LIN {X 0,Y 432.048,Z 691.549,A -85,B 0,C 180,E1 1876.893,E2 1876.893} C_VEL
LIN {X 0,Y 427.007,Z 688.845,A -85,B 0,C 180,E1 1873.962,E2 1873.962} C_VEL
LIN {X 0,Y 421.871,Z 685.398,A -85,B 0,C 180,E1 1871.198,E2 1871.198} C_VEL
LIN {X 0,Y 415.949,Z 680.769,A -85,B 0,C 180,E1 1868.275,E2 1868.275} C_VEL
LIN {X 0,Y 408.852,Z 676.226,A -85,B 0,C 180,E1 1865.437,E2 1865.437} C_VEL
LIN {X 0,Y 401.513,Z 670.583,A -85,B 0,C 180,E1 1862.571,E2 1862.571} C_VEL
LIN {X 0,Y 392.48,Z 664.405,A -85,B 0,C 180,E1 1859.542,E2 1859.542} C_VEL
LIN {X 0,Y 385.757,Z 659.325,A -85,B 0,C 180,E1 1857.38,E2 1857.38} C_VEL
LIN {X 0,Y 377.479,Z 653.334,A -85,B 0,C 180,E1 1854.92,E2 1854.92} C_VEL
LIN {X 0,Y 370.222,Z 647.787,A -85,B 0,C 180,E1 1852.819,E2 1852.819} C_VEL
LIN {X 0,Y 360.53,Z 640.36,A -85,B 0,C 180,E1 1850.166,E2 1850.166} C_VEL
LIN {X 0,Y 343.918,Z 628.074,A -85,B 0,C 180,E1 1845.661,E2 1845.661} C_VEL
LIN {X 0,Y 325.439,Z 613.418,A -85,B 0,C 180,E1 1839.722,E2 1839.722} C_VEL
LIN {X 0,Y 308.556,Z 596.504,A -85,B 0,C 180,E1 1832.543,E2 1832.543} C_VEL
LIN {X 0,Y 297.297,Z 579.607,A -85,B 0,C 180,E1 1825.499,E2 1825.499} C_VEL
LIN {X 0,Y 291.705,Z 565.731,A -85,B 0,C 180,E1 1820.046,E2 1820.046} C_VEL
LIN {X 0,Y 288.211,Z 547.966,A -85,B 0,C 180,E1 1813.697,E2 1813.697} C_VEL
LIN {X 0,Y 287.479,Z 531.833,A -85,B 0,C 180,E1 1808.551,E2 1808.551} C_VEL
LIN {X 0,Y 287.525,Z 526.14,A -85,B 0,C 180,E1 1806.753,E2 1806.753} C_VEL
LIN {X 0,Y 282.899,Z 545.109,A -85,B 0,C 180,E1 1806.656,E2 1806.656} C_VEL
LIN {X 0,Y 277.004,Z 563.845,A -85,B 0,C 180,E1 1806.576,E2 1806.576} C_VEL
LIN {X 0,Y 268.131,Z 586.178,A -85,B 0,C 180,E1 1806.449,E2 1806.449} C_VEL
LIN {X 0,Y 258.493,Z 605.496,A -85,B 0,C 180,E1 1806.291,E2 1806.291} C_VEL
LIN {X 0,Y 248.85,Z 621.951,A -85,B 0,C 180,E1 1806.106,E2 1806.106} C_VEL
LIN {X 0,Y 238.7,Z 637.021,A -85,B 0,C 180,E1 1805.888,E2 1805.888} C_VEL
LIN {X 0,Y 227.028,Z 652.184,A -85,B 0,C 180,E1 1805.601,E2 1805.601} C_VEL
LIN {X 0,Y 211.531,Z 669.665,A -85,B 0,C 180,E1 1805.153,E2 1805.153} C_VEL
LIN {X 0,Y 195.584,Z 684.873,A -85,B 0,C 180,E1 1804.61,E2 1804.61} C_VEL
LIN {X 0,Y 181.403,Z 696.751,A -85,B 0,C 180,E1 1804.026,E2 1804.026} C_VEL
LIN {X 0,Y 167.242,Z 707.237,A -85,B 0,C 180,E1 1803.335,E2 1803.335} C_VEL
LIN {X 0,Y 152.1,Z 717.119,A -85,B 0,C 180,E1 1802.439,E2 1802.439} C_VEL
LIN {X 0,Y 135.999,Z 726.296,A -85,B 0,C 180,E1 1801.251,E2 1801.251} C_VEL
LIN {X 0,Y 116.977,Z 735.612,A -85,B 0,C 180,E1 1799.404,E2 1799.404} C_VEL
LIN {X 0,Y 95.169,Z 744.266,A -85,B 0,C 180,E1 1796.358,E2 1796.358} C_VEL
LIN {X 0,Y 77.459,Z 749.938,A -85,B 0,C 180,E1 1792.583,E2 1792.583} C_VEL
LIN {X 0,Y 61.505,Z 754.079,A -85,B 0,C 180,E1 1787.237,E2 1787.237} C_VEL
LIN {X 0,Y 45.403,Z 757.356,A -85,B 0,C 180,E1 1777.64,E2 1777.64} C_VEL
LIN {X 0,Y 32.323,Z 759.394,A -85,B 0,C 180,E1 1760.647,E2 1760.647} C_VEL
LIN {X 0,Y 24.775,Z 760.386,A -85,B 0,C 180,E1 1731.295,E2 1731.295} C_VEL
LIN {X 0,Y 23.981,Z 760.637,A -85,B 0,C 180,E1 1707.61,E2 1707.61} C_VEL
LIN {X 0,Y 29.264,Z 759.849,A -85,B 0,C 180,E1 1666.9,E2 1666.9} C_VEL
LIN {X 0,Y 43.719,Z 757.656,A -85,B 0,C 180,E1 1643.835,E2 1643.835} C_VEL
LIN {X 0,Y 59.678,Z 754.493,A -85,B 0,C 180,E1 1633.567,E2 1633.567} C_VEL
LIN {X 0,Y 75.698,Z 750.434,A -85,B 0,C 180,E1 1627.892,E2 1627.892} C_VEL
LIN {X 0,Y 92.221,Z 745.27,A -85,B 0,C 180,E1 1624.167,E2 1624.167} C_VEL
LIN {X 0,Y 109.014,Z 738.948,A -85,B 0,C 180,E1 1621.562,E2 1621.562} C_VEL
LIN {X 0,Y 127.974,Z 730.455,A -85,B 0,C 180,E1 1619.46,E2 1619.46} C_VEL
LIN {X 0,Y 149.077,Z 718.975,A -85,B 0,C 180,E1 1617.766,E2 1617.766} C_VEL
LIN {X 0,Y 165.221,Z 708.639,A -85,B 0,C 180,E1 1616.776,E2 1616.776} C_VEL
LIN {X 0,Y 180.391,Z 697.542,A -85,B 0,C 180,E1 1616.019,E2 1616.019} C_VEL
LIN {X 0,Y 193.558,Z 686.651,A -85,B 0,C 180,E1 1615.467,E2 1615.467} C_VEL
LIN {X 0,Y 207.244,Z 673.885,A -85,B 0,C 180,E1 1614.979,E2 1614.979} C_VEL
LIN {X 0,Y 221.286,Z 658.984,A -85,B 0,C 180,E1 1614.555,E2 1614.555} C_VEL
LIN {X 0,Y 236.67,Z 639.862,A -85,B 0,C 180,E1 1614.159,E2 1614.159} C_VEL
LIN {X 0,Y 247.836,Z 623.56,A -85,B 0,C 180,E1 1613.914,E2 1613.914} C_VEL
LIN {X 0,Y 257.478,Z 607.335,A -85,B 0,C 180,E1 1613.727,E2 1613.727} C_VEL
LIN {X 0,Y 266.102,Z 590.426,A -85,B 0,C 180,E1 1613.582,E2 1613.582} C_VEL
LIN {X 0,Y 274.723,Z 570.258,A -85,B 0,C 180,E1 1613.454,E2 1613.454} C_VEL
LIN {X 0,Y 282.17,Z 547.737,A -85,B 0,C 180,E1 1613.355,E2 1613.355} C_VEL
LIN {X 0,Y 287.057,Z 528.29,A -85,B 0,C 180,E1 1613.262,E2 1613.262} C_VEL
LIN {X 0,Y 287.525,Z 526.239,A -85,B 0,C 180,E1 1613.21,E2 1613.21} C_VEL
LIN {X 0,Y 287.819,Z 543.482,A -85,B 0,C 180,E1 1607.765,E2 1607.765} C_VEL
LIN {X 0,Y 288.88,Z 552.893,A -85,B 0,C 180,E1 1604.615,E2 1604.615} C_VEL
LIN {X 0,Y 289.148,Z 557.425,A -85,B 0,C 180,E1 1603.367,E2 1603.367} C_VEL
LIN {X 0,Y 288.555,Z 571.983,A -85,B 0,C 180,E1 1600.311,E2 1600.311} C_VEL
LIN {X 0,Y 288.986,Z 575.602,A -85,B 0,C 180,E1 1599.21,E2 1599.21} C_VEL
LIN {X 0,Y 294.461,Z 588.788,A -85,B 0,C 180,E1 1593.804,E2 1593.804} C_VEL
LIN {X 0,Y 306.56,Z 606.164,A -85,B 0,C 180,E1 1586.264,E2 1586.264} C_VEL
LIN {X 0,Y 326.692,Z 624.896,A -85,B 0,C 180,E1 1578.042,E2 1578.042} C_VEL
LIN {X 0,Y 345.594,Z 639.205,A -85,B 0,C 180,E1 1572.211,E2 1572.211} C_VEL
LIN {X 0,Y 358.052,Z 648.466,A -85,B 0,C 180,E1 1568.819,E2 1568.819} C_VEL
LIN {X 0,Y 367.67,Z 655.59,A -85,B 0,C 180,E1 1566.161,E2 1566.161} C_VEL
LIN {X 0,Y 375.567,Z 661.712,A -85,B 0,C 180,E1 1563.804,E2 1563.804} C_VEL
LIN {X 0,Y 382.824,Z 666.875,A -85,B 0,C 180,E1 1561.628,E2 1561.628} C_VEL
LIN {X 0,Y 391.869,Z 673.574,A -85,B 0,C 180,E1 1558.628,E2 1558.628} C_VEL
LIN {X 0,Y 397.847,Z 677.754,A -85,B 0,C 180,E1 1556.527,E2 1556.527} C_VEL
LIN {X 0,Y 405.855,Z 683.606,A -85,B 0,C 180,E1 1553.366,E2 1553.366} C_VEL
LIN {X 0,Y 411.419,Z 687.152,A -85,B 0,C 180,E1 1551.052,E2 1551.052} C_VEL
LIN {X 0,Y 416.922,Z 691.474,A -85,B 0,C 180,E1 1548.246,E2 1548.246} C_VEL
LIN {X 0,Y 422.748,Z 695.187,A -85,B 0,C 180,E1 1545.078,E2 1545.078} C_VEL
LIN {X 0,Y 427.046,Z 697.466,A -85,B 0,C 180,E1 1542.438,E2 1542.438} C_VEL
LIN {X 0,Y 430.04,Z 700.241,A -85,B 0,C 180,E1 1539.501,E2 1539.501} C_VEL
LIN {X 0,Y 432.467,Z 702.2,A -85,B 0,C 180,E1 1536.504,E2 1536.504} C_VEL
LIN {X 0,Y 434.033,Z 703.321,A -85,B 0,C 180,E1 1533.698,E2 1533.698} C_VEL
LIN {X 0,Y 434.675,Z 703.705,A -85,B 0,C 180,E1 1531.318,E2 1531.318} C_VEL
LIN {X 0,Y 434.753,Z 703.73,A -85,B 0,C 180,E1 1529.209,E2 1529.209} C_VEL
LIN {X 0,Y 434.141,Z 703.379,A -85,B 0,C 180,E1 1526.567,E2 1526.567} C_VEL
LIN {X 0,Y 432.755,Z 702.403,A -85,B 0,C 180,E1 1523.9,E2 1523.9} C_VEL
LIN {X 0,Y 430.41,Z 700.585,A -85,B 0,C 180,E1 1520.912,E2 1520.912} C_VEL
LIN {X 0,Y 427.67,Z 698.099,A -85,B 0,C 180,E1 1518.129,E2 1518.129} C_VEL
LIN {X 0,Y 425.585,Z 696.698,A -85,B 0,C 180,E1 1516.575,E2 1516.575} C_VEL
LIN {X 0,Y 420.846,Z 694.09,A -85,B 0,C 180,E1 1513.863,E2 1513.863} C_VEL
LIN {X 0,Y 415.089,Z 690.135,A -85,B 0,C 180,E1 1510.782,E2 1510.782} C_VEL
LIN {X 0,Y 409.819,Z 686.049,A -85,B 0,C 180,E1 1508.235,E2 1508.235} C_VEL
LIN {X 0,Y 403.522,Z 682.027,A -85,B 0,C 180,E1 1505.715,E2 1505.715} C_VEL
LIN {X 0,Y 396.127,Z 676.336,A -85,B 0,C 180,E1 1502.818,E2 1502.818} C_VEL
LIN {X 0,Y 387.824,Z 670.716,A -85,B 0,C 180,E1 1500.029,E2 1500.029} C_VEL
LIN {X 0,Y 379.753,Z 664.676,A -85,B 0,C 180,E1 1497.412,E2 1497.412} C_VEL
LIN {X 0,Y 370.334,Z 657.748,A -85,B 0,C 180,E1 1494.626,E2 1494.626} C_VEL
LIN {X 0,Y 362.763,Z 652.047,A -85,B 0,C 180,E1 1492.478,E2 1492.478} C_VEL
LIN {X 0,Y 352.04,Z 643.946,A -85,B 0,C 180,E1 1489.57,E2 1489.57} C_VEL
LIN {X 0,Y 337.286,Z 633.069,A -85,B 0,C 180,E1 1485.356,E2 1485.356} C_VEL
LIN {X 0,Y 318.306,Z 617.899,A -85,B 0,C 180,E1 1478.922,E2 1478.922} C_VEL
LIN {X 0,Y 301.774,Z 600.227,A -85,B 0,C 180,E1 1471.124,E2 1471.124} C_VEL
LIN {X 0,Y 291.405,Z 582.303,A -85,B 0,C 180,E1 1463.455,E2 1463.455} C_VEL
LIN {X 0,Y 286.507,Z 564.729,A -85,B 0,C 180,E1 1456.629,E2 1456.629} C_VEL
LIN {X 0,Y 285.15,Z 548.556,A -85,B 0,C 180,E1 1450.979,E2 1450.979} C_VEL
LIN {X 0,Y 285.221,Z 540.34,A -85,B 0,C 180,E1 1448.275,E2 1448.275} C_VEL
LIN {X 0,Y 279.398,Z 559.7,A -85,B 0,C 180,E1 1448.23,E2 1448.23} C_VEL
LIN {X 0,Y 272.99,Z 576.864,A -85,B 0,C 180,E1 1448.187,E2 1448.187} C_VEL
LIN {X 0,Y 265.088,Z 594.503,A -85,B 0,C 180,E1 1448.113,E2 1448.113} C_VEL
LIN {X 0,Y 254.41,Z 614.476,A -85,B 0,C 180,E1 1447.995,E2 1447.995} C_VEL
LIN {X 0,Y 241.969,Z 633.628,A -85,B 0,C 180,E1 1447.838,E2 1447.838} C_VEL
LIN {X 0,Y 230.504,Z 648.864,A -85,B 0,C 180,E1 1447.667,E2 1447.667} C_VEL
LIN {X 0,Y 218.289,Z 663.113,A -85,B 0,C 180,E1 1447.45,E2 1447.45} C_VEL
LIN {X 0,Y 204.038,Z 677.704,A -85,B 0,C 180,E1 1447.155,E2 1447.155} C_VEL
LIN {X 0,Y 185.207,Z 694.205,A -85,B 0,C 180,E1 1446.668,E2 1446.668} C_VEL
LIN {X 0,Y 168.929,Z 706.362,A -85,B 0,C 180,E1 1446.146,E2 1446.146} C_VEL
LIN {X 0,Y 153.68,Z 716.325,A -85,B 0,C 180,E1 1445.542,E2 1445.542} C_VEL
LIN {X 0,Y 138.45,Z 725.037,A -85,B 0,C 180,E1 1444.793,E2 1444.793} C_VEL
LIN {X 0,Y 121.944,Z 733.227,A -85,B 0,C 180,E1 1443.761,E2 1443.761} C_VEL
LIN {X 0,Y 104.055,Z 740.771,A -85,B 0,C 180,E1 1442.262,E2 1442.262} C_VEL
LIN {X 0,Y 81.983,Z 748.355,A -85,B 0,C 180,E1 1439.508,E2 1439.508} C_VEL
LIN {X 0,Y 61.206,Z 753.69,A -85,B 0,C 180,E1 1435.123,E2 1435.123} C_VEL
LIN {X 0,Y 43.904,Z 757.028,A -85,B 0,C 180,E1 1428.282,E2 1428.282} C_VEL
LIN {X 0,Y 28.709,Z 759.125,A -85,B 0,C 180,E1 1414.881,E2 1414.881} C_VEL
LIN {X 0,Y 17.496,Z 760.209,A -85,B 0,C 180,E1 1380.949,E2 1380.949} C_VEL
LIN {X 0,Y 15.972,Z 760.462,A -85,B 0,C 180,E1 1346.411,E2 1346.411} C_VEL
LIN {X 0,Y 25.073,Z 759.54,A -85,B 0,C 180,E1 1291.228,E2 1291.228} C_VEL
LIN {X 0,Y 41.106,Z 757.478,A -85,B 0,C 180,E1 1273.382,E2 1273.382} C_VEL
LIN {X 0,Y 58.278,Z 754.32,A -85,B 0,C 180,E1 1265.744,E2 1265.744} C_VEL
LIN {X 0,Y 75.014,Z 750.256,A -85,B 0,C 180,E1 1261.692,E2 1261.692} C_VEL
LIN {X 0,Y 91.989,Z 745.091,A -85,B 0,C 180,E1 1259.079,E2 1259.079} C_VEL
LIN {X 0,Y 109.097,Z 738.771,A -85,B 0,C 180,E1 1257.266,E2 1257.266} C_VEL
LIN {X 0,Y 128.311,Z 730.279,A -85,B 0,C 180,E1 1255.811,E2 1255.811} C_VEL
LIN {X 0,Y 149.762,Z 718.71,A -85,B 0,C 180,E1 1254.637,E2 1254.637} C_VEL
LIN {X 0,Y 165.878,Z 708.465,A -85,B 0,C 180,E1 1253.966,E2 1253.966} C_VEL
LIN {X 0,Y 181.137,Z 697.367,A -85,B 0,C 180,E1 1253.453,E2 1253.453} C_VEL
LIN {X 0,Y 195.386,Z 685.587,A -85,B 0,C 180,E1 1253.055,E2 1253.055} C_VEL
LIN {X 0,Y 209.636,Z 672.216,A -85,B 0,C 180,E1 1252.726,E2 1252.726} C_VEL
LIN {X 0,Y 225.922,Z 654.529,A -85,B 0,C 180,E1 1252.414,E2 1252.414} C_VEL
LIN {X 0,Y 239.154,Z 637.56,A -85,B 0,C 180,E1 1252.201,E2 1252.201} C_VEL
LIN {X 0,Y 249.836,Z 621.778,A -85,B 0,C 180,E1 1252.056,E2 1252.056} C_VEL
LIN {X 0,Y 259.498,Z 605.326,A -85,B 0,C 180,E1 1251.942,E2 1251.942} C_VEL
LIN {X 0,Y 269.152,Z 586,A -85,B 0,C 180,E1 1251.851,E2 1251.851} C_VEL
LIN {X 0,Y 278.038,Z 563.678,A -85,B 0,C 180,E1 1251.781,E2 1251.781} C_VEL
LIN {X 0,Y 284.004,Z 544.717,A -85,B 0,C 180,E1 1251.736,E2 1251.736} C_VEL
LIN {X 0,Y 285.262,Z 540.289,A -85,B 0,C 180,E1 1251.687,E2 1251.687} C_VEL
LIN {X 0,Y 285.603,Z 557.971,A -85,B 0,C 180,E1 1245.814,E2 1245.814} C_VEL
LIN {X 0,Y 288.188,Z 572.722,A -85,B 0,C 180,E1 1240.333,E2 1240.333} C_VEL
LIN {X 0,Y 288.986,Z 575.602,A -85,B 0,C 180,E1 1239.21,E2 1239.21} C_VEL
LIN {X 0,Y 289.661,Z 579.828,A -85,B 0,C 180,E1 1237.923,E2 1237.923} C_VEL
LIN {X 0,Y 289.945,Z 593.385,A -85,B 0,C 180,E1 1234.696,E2 1234.696} C_VEL
LIN {X 0,Y 290.85,Z 596.648,A -85,B 0,C 180,E1 1233.57,E2 1233.57} C_VEL
LIN {X 0,Y 303.878,Z 614.937,A -85,B 0,C 180,E1 1225.302,E2 1225.302} C_VEL
LIN {X 0,Y 323.118,Z 632.206,A -85,B 0,C 180,E1 1217.425,E2 1217.425} C_VEL
LIN {X 0,Y 340.313,Z 645.101,A -85,B 0,C 180,E1 1211.982,E2 1211.982} C_VEL
LIN {X 0,Y 352.229,Z 653.841,A -85,B 0,C 180,E1 1208.641,E2 1208.641} C_VEL
LIN {X 0,Y 361.939,Z 661.049,A -85,B 0,C 180,E1 1205.959,E2 1205.959} C_VEL
LIN {X 0,Y 370.883,Z 667.919,A -85,B 0,C 180,E1 1203.306,E2 1203.306} C_VEL
LIN {X 0,Y 378.204,Z 673.214,A -85,B 0,C 180,E1 1201.064,E2 1201.064} C_VEL
LIN {X 0,Y 386.833,Z 679.455,A -85,B 0,C 180,E1 1198.185,E2 1198.185} C_VEL
LIN {X 0,Y 392.024,Z 683.129,A -85,B 0,C 180,E1 1196.343,E2 1196.343} C_VEL
LIN {X 0,Y 399.817,Z 688.818,A -85,B 0,C 180,E1 1193.271,E2 1193.271} C_VEL
LIN {X 0,Y 405.586,Z 692.55,A -85,B 0,C 180,E1 1190.876,E2 1190.876} C_VEL
LIN {X 0,Y 411.197,Z 696.903,A -85,B 0,C 180,E1 1187.986,E2 1187.986} C_VEL
LIN {X 0,Y 416.127,Z 700.078,A -85,B 0,C 180,E1 1185.324,E2 1185.324} C_VEL
LIN {X 0,Y 420.877,Z 702.569,A -85,B 0,C 180,E1 1182.465,E2 1182.465} C_VEL
LIN {X 0,Y 423.868,Z 705.347,A -85,B 0,C 180,E1 1179.581,E2 1179.581} C_VEL
LIN {X 0,Y 426.173,Z 707.229,A -85,B 0,C 180,E1 1176.736,E2 1176.736} C_VEL
LIN {X 0,Y 427.744,Z 708.357,A -85,B 0,C 180,E1 1174.021,E2 1174.021} C_VEL
LIN {X 0,Y 428.485,Z 708.783,A -85,B 0,C 180,E1 1171.471,E2 1171.471} C_VEL
LIN {X 0,Y 428.591,Z 708.826,A -85,B 0,C 180,E1 1169.332,E2 1169.332} C_VEL
LIN {X 0,Y 428.064,Z 708.528,A -85,B 0,C 180,E1 1166.787,E2 1166.787} C_VEL
LIN {X 0,Y 426.74,Z 707.626,A -85,B 0,C 180,E1 1164.083,E2 1164.083} C_VEL
LIN {X 0,Y 424.678,Z 706.092,A -85,B 0,C 180,E1 1161.335,E2 1161.335} C_VEL
LIN {X 0,Y 422.103,Z 703.779,A -85,B 0,C 180,E1 1158.663,E2 1158.663} C_VEL
LIN {X 0,Y 419.943,Z 702.077,A -85,B 0,C 180,E1 1156.929,E2 1156.929} C_VEL
LIN {X 0,Y 414.975,Z 699.413,A -85,B 0,C 180,E1 1154.029,E2 1154.029} C_VEL
LIN {X 0,Y 409.055,Z 695.34,A -85,B 0,C 180,E1 1150.883,E2 1150.883} C_VEL
LIN {X 0,Y 404.155,Z 691.495,A -85,B 0,C 180,E1 1148.472,E2 1148.472} C_VEL
LIN {X 0,Y 396.702,Z 686.692,A -85,B 0,C 180,E1 1145.492,E2 1145.492} C_VEL
LIN {X 0,Y 389.268,Z 681.034,A -85,B 0,C 180,E1 1142.631,E2 1142.631} C_VEL
LIN {X 0,Y 380.718,Z 675.133,A -85,B 0,C 180,E1 1139.776,E2 1139.776} C_VEL
LIN {X 0,Y 373.472,Z 669.733,A -85,B 0,C 180,E1 1137.448,E2 1137.448} C_VEL
LIN {X 0,Y 362.618,Z 661.611,A -85,B 0,C 180,E1 1134.233,E2 1134.233} C_VEL
LIN {X 0,Y 353.23,Z 654.62,A -85,B 0,C 180,E1 1131.638,E2 1131.638} C_VEL
LIN {X 0,Y 343.478,Z 647.441,A -85,B 0,C 180,E1 1128.936,E2 1128.936} C_VEL
LIN {X 0,Y 331.052,Z 638.315,A -85,B 0,C 180,E1 1125.217,E2 1125.217} C_VEL
LIN {X 0,Y 313.378,Z 624.206,A -85,B 0,C 180,E1 1118.944,E2 1118.944} C_VEL
LIN {X 0,Y 297.513,Z 607.186,A -85,B 0,C 180,E1 1111.169,E2 1111.169} C_VEL
LIN {X 0,Y 288.151,Z 590.932,A -85,B 0,C 180,E1 1103.953,E2 1103.953} C_VEL
LIN {X 0,Y 283.874,Z 576.6,A -85,B 0,C 180,E1 1098.057,E2 1098.057} C_VEL
LIN {X 0,Y 282.372,Z 561.035,A -85,B 0,C 180,E1 1092.261,E2 1092.261} C_VEL
LIN {X 0,Y 282.538,Z 554.045,A -85,B 0,C 180,E1 1089.857,E2 1089.857} C_VEL
LIN {X 0,Y 274.984,Z 574.891,A -85,B 0,C 180,E1 1089.847,E2 1089.847} C_VEL
LIN {X 0,Y 267.387,Z 592.153,A -85,B 0,C 180,E1 1089.828,E2 1089.828} C_VEL
LIN {X 0,Y 258.203,Z 609.755,A -85,B 0,C 180,E1 1089.797,E2 1089.797} C_VEL
LIN {X 0,Y 245.472,Z 630.284,A -85,B 0,C 180,E1 1089.732,E2 1089.732} C_VEL
LIN {X 0,Y 232.547,Z 647.67,A -85,B 0,C 180,E1 1089.653,E2 1089.653} C_VEL
LIN {X 0,Y 219.995,Z 662.38,A -85,B 0,C 180,E1 1089.55,E2 1089.55} C_VEL
LIN {X 0,Y 206.736,Z 676.035,A -85,B 0,C 180,E1 1089.417,E2 1089.417} C_VEL
LIN {X 0,Y 190.407,Z 690.745,A -85,B 0,C 180,E1 1089.208,E2 1089.208} C_VEL
LIN {X 0,Y 172.034,Z 704.786,A -85,B 0,C 180,E1 1088.911,E2 1088.911} C_VEL
LIN {X 0,Y 155.701,Z 715.531,A -85,B 0,C 180,E1 1088.572,E2 1088.572} C_VEL
LIN {X 0,Y 139.369,Z 724.861,A -85,B 0,C 180,E1 1088.137,E2 1088.137} C_VEL
LIN {X 0,Y 123.045,Z 732.917,A -85,B 0,C 180,E1 1087.58,E2 1087.58} C_VEL
LIN {X 0,Y 105.716,Z 740.196,A -85,B 0,C 180,E1 1086.792,E2 1086.792} C_VEL
LIN {X 0,Y 84.351,Z 747.59,A -85,B 0,C 180,E1 1085.38,E2 1085.38} C_VEL
LIN {X 0,Y 62.066,Z 753.302,A -85,B 0,C 180,E1 1082.94,E2 1082.94} C_VEL
LIN {X 0,Y 43.992,Z 756.699,A -85,B 0,C 180,E1 1079.275,E2 1079.275} C_VEL
LIN {X 0,Y 26.308,Z 758.948,A -85,B 0,C 180,E1 1071.137,E2 1071.137} C_VEL
LIN {X 0,Y 11.352,Z 760.033,A -85,B 0,C 180,E1 1042.433,E2 1042.433} C_VEL
LIN {X 0,Y 7.979,Z 760.286,A -85,B 0,C 180,E1 982.801,E2 982.801} C_VEL
LIN {X 0,Y 21.572,Z 759.403,A -85,B 0,C 180,E1 913.28,E2 913.28} C_VEL
LIN {X 0,Y 40.013,Z 757.3,A -85,B 0,C 180,E1 901.944,E2 901.944} C_VEL
LIN {X 0,Y 58.033,Z 754.142,A -85,B 0,C 180,E1 897.689,E2 897.689} C_VEL
LIN {X 0,Y 75.38,Z 750.035,A -85,B 0,C 180,E1 895.435,E2 895.435} C_VEL
LIN {X 0,Y 92.483,Z 744.914,A -85,B 0,C 180,E1 894.006,E2 894.006} C_VEL
LIN {X 0,Y 109.791,Z 738.595,A -85,B 0,C 180,E1 893.001,E2 893.001} C_VEL
LIN {X 0,Y 130.185,Z 729.636,A -85,B 0,C 180,E1 892.161,E2 892.161} C_VEL
LIN {X 0,Y 150.597,Z 718.623,A -85,B 0,C 180,E1 891.553,E2 891.553} C_VEL
LIN {X 0,Y 166.93,Z 708.291,A -85,B 0,C 180,E1 891.186,E2 891.186} C_VEL
LIN {X 0,Y 182.243,Z 697.193,A -85,B 0,C 180,E1 890.913,E2 890.913} C_VEL
LIN {X 0,Y 196.532,Z 685.413,A -85,B 0,C 180,E1 890.706,E2 890.706} C_VEL
LIN {X 0,Y 211.324,Z 671.544,A -85,B 0,C 180,E1 890.537,E2 890.537} C_VEL
LIN {X 0,Y 228.151,Z 653.098,A -85,B 0,C 180,E1 890.383,E2 890.383} C_VEL
LIN {X 0,Y 240.381,Z 637.389,A -85,B 0,C 180,E1 890.295,E2 890.295} C_VEL
LIN {X 0,Y 251.076,Z 621.605,A -85,B 0,C 180,E1 890.235,E2 890.235} C_VEL
LIN {X 0,Y 260.748,Z 605.157,A -85,B 0,C 180,E1 890.192,E2 890.192} C_VEL
LIN {X 0,Y 270.916,Z 584.717,A -85,B 0,C 180,E1 890.164,E2 890.164} C_VEL
LIN {X 0,Y 279.298,Z 563.512,A -85,B 0,C 180,E1 890.152,E2 890.152} C_VEL
LIN {X 0,Y 282.534,Z 554.12,A -85,B 0,C 180,E1 890.117,E2 890.117} C_VEL
LIN {X 0,Y 283.043,Z 570.679,A -85,B 0,C 180,E1 884.216,E2 884.216} C_VEL
LIN {X 0,Y 286.861,Z 587.688,A -85,B 0,C 180,E1 877.453,E2 877.453} C_VEL
LIN {X 0,Y 290.85,Z 596.648,A -85,B 0,C 180,E1 873.57,E2 873.57} C_VEL
LIN {X 0,Y 292.005,Z 600.459,A -85,B 0,C 180,E1 872.259,E2 872.259} C_VEL
LIN {X 0,Y 293.399,Z 613.038,A -85,B 0,C 180,E1 868.927,E2 868.927} C_VEL
LIN {X 0,Y 294.688,Z 616.052,A -85,B 0,C 180,E1 867.8,E2 867.8} C_VEL
LIN {X 0,Y 310.432,Z 632.147,A -85,B 0,C 180,E1 860.136,E2 860.136} C_VEL
LIN {X 0,Y 330.354,Z 647.449,A -85,B 0,C 180,E1 853.153,E2 853.153} C_VEL
LIN {X 0,Y 346.191,Z 659.013,A -85,B 0,C 180,E1 848.49,E2 848.49} C_VEL
LIN {X 0,Y 357.634,Z 667.595,A -85,B 0,C 180,E1 845.275,E2 845.275} C_VEL
LIN {X 0,Y 367.218,Z 674.688,A -85,B 0,C 180,E1 842.425,E2 842.425} C_VEL
LIN {X 0,Y 373.664,Z 679.47,A -85,B 0,C 180,E1 840.376,E2 840.376} C_VEL
LIN {X 0,Y 382.241,Z 685.519,A -85,B 0,C 180,E1 837.529,E2 837.529} C_VEL
LIN {X 0,Y 387.692,Z 689.585,A -85,B 0,C 180,E1 835.487,E2 835.487} C_VEL
LIN {X 0,Y 394.45,Z 694.342,A -85,B 0,C 180,E1 832.817,E2 832.817} C_VEL
LIN {X 0,Y 399.259,Z 697.441,A -85,B 0,C 180,E1 830.828,E2 830.828} C_VEL
LIN {X 0,Y 405.455,Z 702.241,A -85,B 0,C 180,E1 827.655,E2 827.655} C_VEL
LIN {X 0,Y 410.631,Z 705.454,A -85,B 0,C 180,E1 824.812,E2 824.812} C_VEL
LIN {X 0,Y 414.83,Z 707.765,A -85,B 0,C 180,E1 822.244,E2 822.244} C_VEL
LIN {X 0,Y 417.625,Z 710.319,A -85,B 0,C 180,E1 819.451,E2 819.451} C_VEL
LIN {X 0,Y 419.93,Z 712.167,A -85,B 0,C 180,E1 816.562,E2 816.562} C_VEL
LIN {X 0,Y 421.526,Z 713.296,A -85,B 0,C 180,E1 813.672,E2 813.672} C_VEL
LIN {X 0,Y 422.175,Z 713.693,A -85,B 0,C 180,E1 811.357,E2 811.357} C_VEL
LIN {X 0,Y 422.27,Z 713.73,A -85,B 0,C 180,E1 809.322,E2 809.322} C_VEL
LIN {X 0,Y 421.71,Z 713.409,A -85,B 0,C 180,E1 806.738,E2 806.738} C_VEL
LIN {X 0,Y 420.295,Z 712.427,A -85,B 0,C 180,E1 803.952,E2 803.952} C_VEL
LIN {X 0,Y 418.052,Z 710.708,A -85,B 0,C 180,E1 801.045,E2 801.045} C_VEL
LIN {X 0,Y 415.295,Z 708.228,A -85,B 0,C 180,E1 798.193,E2 798.193} C_VEL
LIN {X 0,Y 413.475,Z 706.951,A -85,B 0,C 180,E1 796.863,E2 796.863} C_VEL
LIN {X 0,Y 408.095,Z 703.97,A -85,B 0,C 180,E1 793.783,E2 793.783} C_VEL
LIN {X 0,Y 402.873,Z 700.336,A -85,B 0,C 180,E1 791.016,E2 791.016} C_VEL
LIN {X 0,Y 397.689,Z 696.359,A -85,B 0,C 180,E1 788.467,E2 788.467} C_VEL
LIN {X 0,Y 389.681,Z 691.103,A -85,B 0,C 180,E1 785.277,E2 785.277} C_VEL
LIN {X 0,Y 382.731,Z 685.845,A -85,B 0,C 180,E1 782.63,E2 782.63} C_VEL
LIN {X 0,Y 373.466,Z 679.331,A -85,B 0,C 180,E1 779.553,E2 779.553} C_VEL
LIN {X 0,Y 367.198,Z 674.684,A -85,B 0,C 180,E1 777.564,E2 777.564} C_VEL
LIN {X 0,Y 356.044,Z 666.298,A -85,B 0,C 180,E1 774.254,E2 774.254} C_VEL
LIN {X 0,Y 341.877,Z 655.789,A -85,B 0,C 180,E1 770.282,E2 770.282} C_VEL
LIN {X 0,Y 326.257,Z 644.595,A -85,B 0,C 180,E1 765.568,E2 765.568} C_VEL
LIN {X 0,Y 308.273,Z 630.366,A -85,B 0,C 180,E1 758.994,E2 758.994} C_VEL
LIN {X 0,Y 292.262,Z 612.853,A -85,B 0,C 180,E1 750.648,E2 750.648} C_VEL
LIN {X 0,Y 283.132,Z 595.381,A -85,B 0,C 180,E1 742.64,E2 742.64} C_VEL
LIN {X 0,Y 279.644,Z 578.773,A -85,B 0,C 180,E1 735.768,E2 735.768} C_VEL
LIN {X 0,Y 279.386,Z 567.375,A -85,B 0,C 180,E1 731.473,E2 731.473} C_VEL
LIN {X 0,Y 270.371,Z 588.861,A -85,B 0,C 180,E1 731.51,E2 731.51} C_VEL
LIN {X 0,Y 261.221,Z 606.827,A -85,B 0,C 180,E1 731.544,E2 731.544} C_VEL
LIN {X 0,Y 251.549,Z 623.044,A -85,B 0,C 180,E1 731.569,E2 731.569} C_VEL
LIN {X 0,Y 238.814,Z 641.465,A -85,B 0,C 180,E1 731.593,E2 731.593} C_VEL
LIN {X 0,Y 223.52,Z 659.968,A -85,B 0,C 180,E1 731.612,E2 731.612} C_VEL
LIN {X 0,Y 210.255,Z 673.867,A -85,B 0,C 180,E1 731.616,E2 731.616} C_VEL
LIN {X 0,Y 196.983,Z 686.128,A -85,B 0,C 180,E1 731.611,E2 731.611} C_VEL
LIN {X 0,Y 182.679,Z 697.81,A -85,B 0,C 180,E1 731.588,E2 731.588} C_VEL
LIN {X 0,Y 164.962,Z 710.452,A -85,B 0,C 180,E1 731.538,E2 731.538} C_VEL
LIN {X 0,Y 143.824,Z 723.061,A -85,B 0,C 180,E1 731.444,E2 731.444} C_VEL
LIN {X 0,Y 126.432,Z 731.804,A -85,B 0,C 180,E1 731.329,E2 731.329} C_VEL
LIN {X 0,Y 109.038,Z 739.22,A -85,B 0,C 180,E1 731.166,E2 731.166} C_VEL
LIN {X 0,Y 91.645,Z 745.407,A -85,B 0,C 180,E1 730.945,E2 730.945} C_VEL
LIN {X 0,Y 72.214,Z 750.987,A -85,B 0,C 180,E1 730.598,E2 730.598} C_VEL
LIN {X 0,Y 47.702,Z 756.073,A -85,B 0,C 180,E1 729.922,E2 729.922} C_VEL
LIN {X 0,Y 28.346,Z 758.589,A -85,B 0,C 180,E1 729.051,E2 729.051} C_VEL
LIN {X 0,Y 10.084,Z 759.824,A -85,B 0,C 180,E1 727.516,E2 727.516} C_VEL
LIN {X 0,Y 1.007,Z 760.111,A -85,B 0,C 180,E1 893.396,E2 893.396} C_VEL
LIN {X 0,Y 22.248,Z 759.135,A -85,B 0,C 180,E1 891.345,E2 891.345} C_VEL
LIN {X 0,Y 41.583,Z 756.974,A -85,B 0,C 180,E1 890.31,E2 890.31} C_VEL
LIN {X 0,Y 59.952,Z 753.757,A -85,B 0,C 180,E1 889.696,E2 889.696} C_VEL
LIN {X 0,Y 78.349,Z 749.359,A -85,B 0,C 180,E1 889.278,E2 889.278} C_VEL
LIN {X 0,Y 99.144,Z 742.954,A -85,B 0,C 180,E1 888.953,E2 888.953} C_VEL
LIN {X 0,Y 121.317,Z 734.148,A -85,B 0,C 180,E1 888.714,E2 888.714} C_VEL
LIN {X 0,Y 138.71,Z 725.768,A -85,B 0,C 180,E1 888.585,E2 888.585} C_VEL
LIN {X 0,Y 155.415,Z 716.388,A -85,B 0,C 180,E1 888.496,E2 888.496} C_VEL
LIN {X 0,Y 171.437,Z 706.014,A -85,B 0,C 180,E1 888.439,E2 888.439} C_VEL
LIN {X 0,Y 188.999,Z 692.918,A -85,B 0,C 180,E1 888.402,E2 888.402} C_VEL
LIN {X 0,Y 207.194,Z 676.86,A -85,B 0,C 180,E1 888.383,E2 888.383} C_VEL
LIN {X 0,Y 220.971,Z 662.767,A -85,B 0,C 180,E1 888.386,E2 888.386} C_VEL
LIN {X 0,Y 233.637,Z 647.992,A -85,B 0,C 180,E1 888.396,E2 888.396} C_VEL
LIN {X 0,Y 246.454,Z 630.827,A -85,B 0,C 180,E1 888.423,E2 888.423} C_VEL
LIN {X 0,Y 259.183,Z 610.505,A -85,B 0,C 180,E1 888.452,E2 888.452} C_VEL
LIN {X 0,Y 268.672,Z 592.408,A -85,B 0,C 180,E1 888.484,E2 888.484} C_VEL
LIN {X 0,Y 276.104,Z 575.619,A -85,B 0,C 180,E1 888.511,E2 888.511} C_VEL
LIN {X 0,Y 279.384,Z 567.474,A -85,B 0,C 180,E1 888.492,E2 888.492} C_VEL
LIN {X 0,Y 280.519,Z 585.053,A -85,B 0,C 180,E1 881.719,E2 881.719} C_VEL
LIN {X 0,Y 284.374,Z 598.537,A -85,B 0,C 180,E1 875.929,E2 875.929} C_VEL
LIN {X 0,Y 294.048,Z 615.245,A -85,B 0,C 180,E1 868.192,E2 868.192} C_VEL
LIN {X 0,Y 294.688,Z 616.052,A -85,B 0,C 180,E1 867.8,E2 867.8} C_VEL
LIN {X 0,Y 296.333,Z 619.595,A -85,B 0,C 180,E1 866.495,E2 866.495} C_VEL
LIN {X 0,Y 298.816,Z 631.447,A -85,B 0,C 180,E1 863.134,E2 863.134} C_VEL
LIN {X 0,Y 300.612,Z 634.258,A -85,B 0,C 180,E1 862.034,E2 862.034} C_VEL
LIN {X 0,Y 319.868,Z 649.674,A -85,B 0,C 180,E1 854.544,E2 854.544} C_VEL
LIN {X 0,Y 333.176,Z 659.171,A -85,B 0,C 180,E1 850.335,E2 850.335} C_VEL
LIN {X 0,Y 343.924,Z 666.91,A -85,B 0,C 180,E1 847.193,E2 847.193} C_VEL
LIN {X 0,Y 352.12,Z 673.006,A -85,B 0,C 180,E1 844.85,E2 844.85} C_VEL
LIN {X 0,Y 361.332,Z 679.81,A -85,B 0,C 180,E1 842.137,E2 842.137} C_VEL
LIN {X 0,Y 369.19,Z 685.669,A -85,B 0,C 180,E1 839.613,E2 839.613} C_VEL
LIN {X 0,Y 377.769,Z 691.5,A -85,B 0,C 180,E1 836.737,E2 836.737} C_VEL
LIN {X 0,Y 384.517,Z 696.695,A -85,B 0,C 180,E1 834.092,E2 834.092} C_VEL
LIN {X 0,Y 391.209,Z 701.038,A -85,B 0,C 180,E1 831.435,E2 831.435} C_VEL
LIN {X 0,Y 396.387,Z 705.014,A -85,B 0,C 180,E1 828.925,E2 828.925} C_VEL
LIN {X 0,Y 401.8,Z 708.747,A -85,B 0,C 180,E1 826.033,E2 826.033} C_VEL
LIN {X 0,Y 406.793,Z 711.563,A -85,B 0,C 180,E1 823.212,E2 823.212} C_VEL
LIN {X 0,Y 408.835,Z 712.906,A -85,B 0,C 180,E1 821.71,E2 821.71} C_VEL
LIN {X 0,Y 411.536,Z 715.352,A -85,B 0,C 180,E1 818.944,E2 818.944} C_VEL
LIN {X 0,Y 413.86,Z 717.156,A -85,B 0,C 180,E1 815.962,E2 815.962} C_VEL
LIN {X 0,Y 415.173,Z 718.056,A -85,B 0,C 180,E1 813.313,E2 813.313} C_VEL
LIN {X 0,Y 415.755,Z 718.417,A -85,B 0,C 180,E1 810.965,E2 810.965} C_VEL
LIN {X 0,Y 415.7,Z 718.4,A -85,B 0,C 180,E1 808.346,E2 808.346} C_VEL
LIN {X 0,Y 414.742,Z 717.781,A -85,B 0,C 180,E1 805.576,E2 805.576} C_VEL
LIN {X 0,Y 412.941,Z 716.495,A -85,B 0,C 180,E1 802.768,E2 802.768} C_VEL
LIN {X 0,Y 410.349,Z 714.267,A -85,B 0,C 180,E1 799.755,E2 799.755} C_VEL
LIN {X 0,Y 407.539,Z 711.93,A -85,B 0,C 180,E1 797.245,E2 797.245} C_VEL
LIN {X 0,Y 402.991,Z 709.491,A -85,B 0,C 180,E1 794.606,E2 794.606} C_VEL
LIN {X 0,Y 397.25,Z 705.676,A -85,B 0,C 180,E1 791.512,E2 791.512} C_VEL
LIN {X 0,Y 391.631,Z 701.294,A -85,B 0,C 180,E1 788.733,E2 788.733} C_VEL
LIN {X 0,Y 384.996,Z 697.045,A -85,B 0,C 180,E1 786.092,E2 786.092} C_VEL
LIN {X 0,Y 377.788,Z 691.523,A -85,B 0,C 180,E1 783.264,E2 783.264} C_VEL
LIN {X 0,Y 368.681,Z 685.3,A -85,B 0,C 180,E1 780.212,E2 780.212} C_VEL
LIN {X 0,Y 361.337,Z 679.816,A -85,B 0,C 180,E1 777.862,E2 777.862} C_VEL
LIN {X 0,Y 351.352,Z 672.399,A -85,B 0,C 180,E1 774.916,E2 774.916} C_VEL
LIN {X 0,Y 339.069,Z 663.303,A -85,B 0,C 180,E1 771.395,E2 771.395} C_VEL
LIN {X 0,Y 321.874,Z 651.111,A -85,B 0,C 180,E1 766.112,E2 766.112} C_VEL
LIN {X 0,Y 303.066,Z 636.435,A -85,B 0,C 180,E1 759.062,E2 759.062} C_VEL
LIN {X 0,Y 288.556,Z 620.792,A -85,B 0,C 180,E1 751.317,E2 751.317} C_VEL
LIN {X 0,Y 280.329,Z 606.015,A -85,B 0,C 180,E1 744.217,E2 744.217} C_VEL
LIN {X 0,Y 276.93,Z 593.834,A -85,B 0,C 180,E1 738.744,E2 738.744} C_VEL
LIN {X 0,Y 275.84,Z 580.284,A -85,B 0,C 180,E1 733.132,E2 733.132} C_VEL
LIN {X 0,Y 264.98,Z 602.98,A -85,B 0,C 180,E1 733.241,E2 733.241} C_VEL
LIN {X 0,Y 254.813,Z 620.456,A -85,B 0,C 180,E1 733.339,E2 733.339} C_VEL
LIN {X 0,Y 244.129,Z 636.338,A -85,B 0,C 180,E1 733.442,E2 733.442} C_VEL
LIN {X 0,Y 231.4,Z 652.753,A -85,B 0,C 180,E1 733.566,E2 733.566} C_VEL
LIN {X 0,Y 214.867,Z 670.92,A -85,B 0,C 180,E1 733.729,E2 733.729} C_VEL
LIN {X 0,Y 199.796,Z 685.064,A -85,B 0,C 180,E1 733.892,E2 733.892} C_VEL
LIN {X 0,Y 185.313,Z 696.993,A -85,B 0,C 180,E1 734.052,E2 734.052} C_VEL
LIN {X 0,Y 169.165,Z 708.643,A -85,B 0,C 180,E1 734.251,E2 734.251} C_VEL
LIN {X 0,Y 148.727,Z 721.256,A -85,B 0,C 180,E1 734.54,E2 734.54} C_VEL
LIN {X 0,Y 129.309,Z 731.16,A -85,B 0,C 180,E1 734.886,E2 734.886} C_VEL
LIN {X 0,Y 111.933,Z 738.644,A -85,B 0,C 180,E1 735.286,E2 735.286} C_VEL
LIN {X 0,Y 94.565,Z 744.895,A -85,B 0,C 180,E1 735.832,E2 735.832} C_VEL
LIN {X 0,Y 76.691,Z 750.135,A -85,B 0,C 180,E1 736.668,E2 736.668} C_VEL
LIN {X 0,Y 55.844,Z 754.841,A -85,B 0,C 180,E1 738.407,E2 738.407} C_VEL
LIN {X 0,Y 31.69,Z 758.322,A -85,B 0,C 180,E1 743.809,E2 743.809} C_VEL
LIN {X 0,Y 14.58,Z 759.616,A -85,B 0,C 180,E1 761.04,E2 761.04} C_VEL
LIN {X 0,Y 8.217,Z 759.937,A -85,B 0,C 180,E1 816.989,E2 816.989} C_VEL
LIN {X 0,Y 24.81,Z 758.96,A -85,B 0,C 180,E1 872.439,E2 872.439} C_VEL
LIN {X 0,Y 43.704,Z 756.799,A -85,B 0,C 180,E1 879.703,E2 879.703} C_VEL
LIN {X 0,Y 61.939,Z 753.581,A -85,B 0,C 180,E1 882.234,E2 882.234} C_VEL
LIN {X 0,Y 80.274,Z 749.182,A -85,B 0,C 180,E1 883.532,E2 883.532} C_VEL
LIN {X 0,Y 101.714,Z 742.553,A -85,B 0,C 180,E1 884.419,E2 884.419} C_VEL
LIN {X 0,Y 123.572,Z 733.791,A -85,B 0,C 180,E1 884.994,E2 884.994} C_VEL
LIN {X 0,Y 141.575,Z 725.05,A -85,B 0,C 180,E1 885.341,E2 885.341} C_VEL
LIN {X 0,Y 157.927,Z 715.798,A -85,B 0,C 180,E1 885.596,E2 885.596} C_VEL
LIN {X 0,Y 175.292,Z 704.438,A -85,B 0,C 180,E1 885.829,E2 885.829} C_VEL
LIN {X 0,Y 195.072,Z 689.177,A -85,B 0,C 180,E1 886.06,E2 886.06} C_VEL
LIN {X 0,Y 210.505,Z 675.191,A -85,B 0,C 180,E1 886.224,E2 886.224} C_VEL
LIN {X 0,Y 223.759,Z 661.474,A -85,B 0,C 180,E1 886.358,E2 886.358} C_VEL
LIN {X 0,Y 237.005,Z 645.829,A -85,B 0,C 180,E1 886.486,E2 886.486} C_VEL
LIN {X 0,Y 251.252,Z 626.091,A -85,B 0,C 180,E1 886.627,E2 886.627} C_VEL
LIN {X 0,Y 261.932,Z 608.497,A -85,B 0,C 180,E1 886.729,E2 886.729} C_VEL
LIN {X 0,Y 271.074,Z 590.815,A -85,B 0,C 180,E1 886.821,E2 886.821} C_VEL
LIN {X 0,Y 275.919,Z 580.123,A -85,B 0,C 180,E1 886.856,E2 886.856} C_VEL
LIN {X 0,Y 277.302,Z 595.86,A -85,B 0,C 180,E1 880.407,E2 880.407} C_VEL
LIN {X 0,Y 282.926,Z 611.747,A -85,B 0,C 180,E1 873.104,E2 873.104} C_VEL
LIN {X 0,Y 295.744,Z 629.373,A -85,B 0,C 180,E1 864.442,E2 864.442} C_VEL
LIN {X 0,Y 300.612,Z 634.258,A -85,B 0,C 180,E1 862.034,E2 862.034} C_VEL
LIN {X 0,Y 302.824,Z 637.506,A -85,B 0,C 180,E1 860.763,E2 860.763} C_VEL
LIN {X 0,Y 306.879,Z 648.959,A -85,B 0,C 180,E1 857.239,E2 857.239} C_VEL
LIN {X 0,Y 308.785,Z 651.131,A -85,B 0,C 180,E1 856.357,E2 856.357} C_VEL
LIN {X 0,Y 324.477,Z 662.482,A -85,B 0,C 180,E1 850.976,E2 850.976} C_VEL
LIN {X 0,Y 335.356,Z 670.096,A -85,B 0,C 180,E1 847.672,E2 847.672} C_VEL
LIN {X 0,Y 345.49,Z 677.478,A -85,B 0,C 180,E1 844.721,E2 844.721} C_VEL
LIN {X 0,Y 356.648,Z 685.603,A -85,B 0,C 180,E1 841.426,E2 841.426} C_VEL
LIN {X 0,Y 365.37,Z 692.13,A -85,B 0,C 180,E1 838.542,E2 838.542} C_VEL
LIN {X 0,Y 372.734,Z 697.245,A -85,B 0,C 180,E1 836.016,E2 836.016} C_VEL
LIN {X 0,Y 381.327,Z 703.499,A -85,B 0,C 180,E1 832.632,E2 832.632} C_VEL
LIN {X 0,Y 386.588,Z 706.906,A -85,B 0,C 180,E1 830.434,E2 830.434} C_VEL
LIN {X 0,Y 391.943,Z 711.032,A -85,B 0,C 180,E1 827.67,E2 827.67} C_VEL
LIN {X 0,Y 397.405,Z 714.534,A -85,B 0,C 180,E1 824.719,E2 824.719} C_VEL
LIN {X 0,Y 401.782,Z 716.938,A -85,B 0,C 180,E1 822.03,E2 822.03} C_VEL
LIN {X 0,Y 404.722,Z 719.644,A -85,B 0,C 180,E1 819.096,E2 819.096} C_VEL
LIN {X 0,Y 406.875,Z 721.327,A -85,B 0,C 180,E1 816.348,E2 816.348} C_VEL
LIN {X 0,Y 408.363,Z 722.337,A -85,B 0,C 180,E1 813.509,E2 813.509} C_VEL
LIN {X 0,Y 408.972,Z 722.71,A -85,B 0,C 180,E1 811.261,E2 811.261} C_VEL
LIN {X 0,Y 409.043,Z 722.733,A -85,B 0,C 180,E1 809.16,E2 809.16} C_VEL
LIN {X 0,Y 408.387,Z 722.359,A -85,B 0,C 180,E1 806.491,E2 806.491} C_VEL
LIN {X 0,Y 406.975,Z 721.388,A -85,B 0,C 180,E1 803.795,E2 803.795} C_VEL
LIN {X 0,Y 404.836,Z 719.74,A -85,B 0,C 180,E1 801.05,E2 801.05} C_VEL
LIN {X 0,Y 402.055,Z 717.208,A -85,B 0,C 180,E1 798.235,E2 798.235} C_VEL
LIN {X 0,Y 399.758,Z 715.773,A -85,B 0,C 180,E1 796.652,E2 796.652} C_VEL
LIN {X 0,Y 394.748,Z 712.938,A -85,B 0,C 180,E1 793.824,E2 793.824} C_VEL
LIN {X 0,Y 388.691,Z 708.629,A -85,B 0,C 180,E1 790.622,E2 790.622} C_VEL
LIN {X 0,Y 384.432,Z 705.421,A -85,B 0,C 180,E1 788.614,E2 788.614} C_VEL
LIN {X 0,Y 377.23,Z 700.674,A -85,B 0,C 180,E1 785.757,E2 785.757} C_VEL
LIN {X 0,Y 370.698,Z 695.688,A -85,B 0,C 180,E1 783.229,E2 783.229} C_VEL
LIN {X 0,Y 361.691,Z 689.458,A -85,B 0,C 180,E1 780.233,E2 780.233} C_VEL
LIN {X 0,Y 354.673,Z 684.255,A -85,B 0,C 180,E1 777.999,E2 777.999} C_VEL
LIN {X 0,Y 344.188,Z 676.427,A -85,B 0,C 180,E1 774.892,E2 774.892} C_VEL
LIN {X 0,Y 329.222,Z 665.705,A -85,B 0,C 180,E1 770.483,E2 770.483} C_VEL
LIN {X 0,Y 314.86,Z 655.7,A -85,B 0,C 180,E1 765.865,E2 765.865} C_VEL
LIN {X 0,Y 297.718,Z 642.376,A -85,B 0,C 180,E1 759.131,E2 759.131} C_VEL
LIN {X 0,Y 282.222,Z 625.099,A -85,B 0,C 180,E1 750.191,E2 750.191} C_VEL
LIN {X 0,Y 274.451,Z 608.589,A -85,B 0,C 180,E1 742.04,E2 742.04} C_VEL
LIN {X 0,Y 272.21,Z 593.048,A -85,B 0,C 180,E1 735.117,E2 735.117} C_VEL
LIN {X 0,Y 272.198,Z 592.378,A -85,B 0,C 180,E1 734.84,E2 734.84} C_VEL
LIN {X 0,Y 262.371,Z 611.087,A -85,B 0,C 180,E1 734.995,E2 734.995} C_VEL
LIN {X 0,Y 249.175,Z 631.907,A -85,B 0,C 180,E1 735.216,E2 735.216} C_VEL
LIN {X 0,Y 236.48,Z 648.804,A -85,B 0,C 180,E1 735.442,E2 735.442} C_VEL
LIN {X 0,Y 223.769,Z 663.541,A -85,B 0,C 180,E1 735.676,E2 735.676} C_VEL
LIN {X 0,Y 208.001,Z 679.47,A -85,B 0,C 180,E1 735.993,E2 735.993} C_VEL
LIN {X 0,Y 190.697,Z 694.299,A -85,B 0,C 180,E1 736.383,E2 736.383} C_VEL
LIN {X 0,Y 174.405,Z 706.367,A -85,B 0,C 180,E1 736.804,E2 736.804} C_VEL
LIN {X 0,Y 158.065,Z 716.888,A -85,B 0,C 180,E1 737.296,E2 737.296} C_VEL
LIN {X 0,Y 138.765,Z 727.582,A -85,B 0,C 180,E1 738.008,E2 738.008} C_VEL
LIN {X 0,Y 117.407,Z 737.268,A -85,B 0,C 180,E1 739.057,E2 739.057} C_VEL
LIN {X 0,Y 99.141,Z 744.049,A -85,B 0,C 180,E1 740.31,E2 740.31} C_VEL
LIN {X 0,Y 80.949,Z 749.548,A -85,B 0,C 180,E1 742.137,E2 742.137} C_VEL
LIN {X 0,Y 62.91,Z 753.825,A -85,B 0,C 180,E1 745.064,E2 745.064} C_VEL
LIN {X 0,Y 42.348,Z 757.374,A -85,B 0,C 180,E1 751.801,E2 751.801} C_VEL
LIN {X 0,Y 22.146,Z 759.378,A -85,B 0,C 180,E1 774.36,E2 774.36} C_VEL
LIN {X 0,Y 16.094,Z 759.78,A -85,B 0,C 180,E1 810,E2 810} C_VEL
LIN {X 0,Y 29.469,Z 758.785,A -85,B 0,C 180,E1 858.276,E2 858.276} C_VEL
LIN {X 0,Y 47.161,Z 756.623,A -85,B 0,C 180,E1 870.36,E2 870.36} C_VEL
LIN {X 0,Y 64.903,Z 753.405,A -85,B 0,C 180,E1 875.344,E2 875.344} C_VEL
LIN {X 0,Y 83.249,Z 748.928,A -85,B 0,C 180,E1 878.14,E2 878.14} C_VEL
LIN {X 0,Y 105.222,Z 742.032,A -85,B 0,C 180,E1 880.159,E2 880.159} C_VEL
LIN {X 0,Y 126.558,Z 733.329,A -85,B 0,C 180,E1 881.432,E2 881.432} C_VEL
LIN {X 0,Y 143.901,Z 724.851,A -85,B 0,C 180,E1 882.198,E2 882.198} C_VEL
LIN {X 0,Y 160.147,Z 715.622,A -85,B 0,C 180,E1 882.772,E2 882.772} C_VEL
LIN {X 0,Y 177.458,Z 704.264,A -85,B 0,C 180,E1 883.283,E2 883.283} C_VEL
LIN {X 0,Y 196.804,Z 689.334,A -85,B 0,C 180,E1 883.762,E2 883.762} C_VEL
LIN {X 0,Y 212.579,Z 675.018,A -85,B 0,C 180,E1 884.103,E2 884.103} C_VEL
LIN {X 0,Y 226.311,Z 660.741,A -85,B 0,C 180,E1 884.373,E2 884.373} C_VEL
LIN {X 0,Y 240.542,Z 643.768,A -85,B 0,C 180,E1 884.633,E2 884.633} C_VEL
LIN {X 0,Y 254.253,Z 624.308,A -85,B 0,C 180,E1 884.87,E2 884.87} C_VEL
LIN {X 0,Y 264.403,Z 607.408,A -85,B 0,C 180,E1 885.036,E2 885.036} C_VEL
LIN {X 0,Y 272.198,Z 592.435,A -85,B 0,C 180,E1 885.137,E2 885.137} C_VEL
LIN {X 0,Y 274.186,Z 607.686,A -85,B 0,C 180,E1 878.388,E2 878.388} C_VEL
LIN {X 0,Y 281.437,Z 623.903,A -85,B 0,C 180,E1 870.407,E2 870.407} C_VEL
LIN {X 0,Y 295.734,Z 640.641,A -85,B 0,C 180,E1 861.776,E2 861.776} C_VEL
LIN {X 0,Y 308.785,Z 651.131,A -85,B 0,C 180,E1 856.357,E2 856.357} C_VEL
LIN {X 0,Y 311.328,Z 654.311,A -85,B 0,C 180,E1 855.132,E2 855.132} C_VEL
LIN {X 0,Y 315.751,Z 664.89,A -85,B 0,C 180,E1 851.853,E2 851.853} C_VEL
LIN {X 0,Y 318.229,Z 667.453,A -85,B 0,C 180,E1 850.836,E2 850.836} C_VEL
LIN {X 0,Y 329.202,Z 674.96,A -85,B 0,C 180,E1 847.4,E2 847.4} C_VEL
LIN {X 0,Y 339.261,Z 682.107,A -85,B 0,C 180,E1 844.388,E2 844.388} C_VEL
LIN {X 0,Y 350.411,Z 690.182,A -85,B 0,C 180,E1 841.092,E2 841.092} C_VEL
LIN {X 0,Y 359.94,Z 697.282,A -85,B 0,C 180,E1 837.946,E2 837.946} C_VEL
LIN {X 0,Y 365.818,Z 701.304,A -85,B 0,C 180,E1 835.93,E2 835.93} C_VEL
LIN {X 0,Y 373.456,Z 706.958,A -85,B 0,C 180,E1 832.923,E2 832.923} C_VEL
LIN {X 0,Y 379.795,Z 711.086,A -85,B 0,C 180,E1 830.333,E2 830.333} C_VEL
LIN {X 0,Y 386.234,Z 715.995,A -85,B 0,C 180,E1 827.007,E2 827.007} C_VEL
LIN {X 0,Y 391.914,Z 719.422,A -85,B 0,C 180,E1 823.874,E2 823.874} C_VEL
LIN {X 0,Y 395.124,Z 721.265,A -85,B 0,C 180,E1 821.826,E2 821.826} C_VEL
LIN {X 0,Y 397.802,Z 723.689,A -85,B 0,C 180,E1 819.11,E2 819.11} C_VEL
LIN {X 0,Y 400.201,Z 725.554,A -85,B 0,C 180,E1 816.023,E2 816.023} C_VEL
LIN {X 0,Y 401.571,Z 726.481,A -85,B 0,C 180,E1 813.283,E2 813.283} C_VEL
LIN {X 0,Y 402.153,Z 726.847,A -85,B 0,C 180,E1 810.997,E2 810.997} C_VEL
LIN {X 0,Y 402.12,Z 726.84,A -85,B 0,C 180,E1 808.433,E2 808.433} C_VEL
LIN {X 0,Y 401.14,Z 726.209,A -85,B 0,C 180,E1 805.599,E2 805.599} C_VEL
LIN {X 0,Y 399.366,Z 724.961,A -85,B 0,C 180,E1 802.81,E2 802.81} C_VEL
LIN {X 0,Y 396.865,Z 722.856,A -85,B 0,C 180,E1 799.843,E2 799.843} C_VEL
LIN {X 0,Y 394.268,Z 720.647,A -85,B 0,C 180,E1 797.525,E2 797.525} C_VEL
LIN {X 0,Y 389.001,Z 717.77,A -85,B 0,C 180,E1 794.497,E2 794.497} C_VEL
LIN {X 0,Y 383.566,Z 714.058,A -85,B 0,C 180,E1 791.602,E2 791.602} C_VEL
LIN {X 0,Y 378.597,Z 710.214,A -85,B 0,C 180,E1 789.115,E2 789.115} C_VEL
LIN {X 0,Y 370.373,Z 704.826,A -85,B 0,C 180,E1 785.853,E2 785.853} C_VEL
LIN {X 0,Y 363.728,Z 699.81,A -85,B 0,C 180,E1 783.308,E2 783.308} C_VEL
LIN {X 0,Y 354.074,Z 693.019,A -85,B 0,C 180,E1 780.107,E2 780.107} C_VEL
LIN {X 0,Y 347.415,Z 688.141,A -85,B 0,C 180,E1 778.029,E2 778.029} C_VEL
LIN {X 0,Y 334.287,Z 678.501,A -85,B 0,C 180,E1 774.114,E2 774.114} C_VEL
LIN {X 0,Y 322.007,Z 670.011,A -85,B 0,C 180,E1 770.362,E2 770.362} C_VEL
LIN {X 0,Y 308.316,Z 660.597,A -85,B 0,C 180,E1 765.784,E2 765.784} C_VEL
LIN {X 0,Y 289.162,Z 645.454,A -85,B 0,C 180,E1 757.738,E2 757.738} C_VEL
LIN {X 0,Y 276.142,Z 629.688,A -85,B 0,C 180,E1 749.247,E2 749.247} C_VEL
LIN {X 0,Y 269.409,Z 612.858,A -85,B 0,C 180,E1 740.646,E2 740.646} C_VEL
LIN {X 0,Y 268.236,Z 604.251,A -85,B 0,C 180,E1 736.597,E2 736.597} C_VEL
LIN {X 0,Y 258.498,Z 620.916,A -85,B 0,C 180,E1 736.82,E2 736.82} C_VEL
LIN {X 0,Y 247.191,Z 637.655,A -85,B 0,C 180,E1 737.092,E2 737.092} C_VEL
LIN {X 0,Y 232.672,Z 656.062,A -85,B 0,C 180,E1 737.466,E2 737.466} C_VEL
LIN {X 0,Y 217.472,Z 672.352,A -85,B 0,C 180,E1 737.897,E2 737.897} C_VEL
LIN {X 0,Y 203.285,Z 685.604,A -85,B 0,C 180,E1 738.347,E2 738.347} C_VEL
LIN {X 0,Y 188.076,Z 698.078,A -85,B 0,C 180,E1 738.882,E2 738.882} C_VEL
LIN {X 0,Y 168.82,Z 711.728,A -85,B 0,C 180,E1 739.679,E2 739.679} C_VEL
LIN {X 0,Y 149.589,Z 723.075,A -85,B 0,C 180,E1 740.664,E2 740.664} C_VEL
LIN {X 0,Y 132.416,Z 731.748,A -85,B 0,C 180,E1 741.773,E2 741.773} C_VEL
LIN {X 0,Y 114.292,Z 739.493,A -85,B 0,C 180,E1 743.297,E2 743.297} C_VEL
LIN {X 0,Y 92.297,Z 747.186,A -85,B 0,C 180,E1 745.967,E2 745.967} C_VEL
LIN {X 0,Y 70.654,Z 752.809,A -85,B 0,C 180,E1 750.328,E2 750.328} C_VEL
LIN {X 0,Y 52.608,Z 756.298,A -85,B 0,C 180,E1 757.045,E2 757.045} C_VEL
LIN {X 0,Y 36.426,Z 758.49,A -85,B 0,C 180,E1 770.228,E2 770.228} C_VEL
LIN {X 0,Y 25.005,Z 759.491,A -85,B 0,C 180,E1 800.798,E2 800.798} C_VEL
LIN {X 0,Y 24.286,Z 759.585,A -85,B 0,C 180,E1 812.36,E2 812.36} C_VEL
LIN {X 0,Y 35.41,Z 758.61,A -85,B 0,C 180,E1 848.4,E2 848.4} C_VEL
LIN {X 0,Y 51.688,Z 756.448,A -85,B 0,C 180,E1 862.469,E2 862.469} C_VEL
LIN {X 0,Y 68.717,Z 753.229,A -85,B 0,C 180,E1 869.136,E2 869.136} C_VEL
LIN {X 0,Y 86.348,Z 748.828,A -85,B 0,C 180,E1 873.065,E2 873.065} C_VEL
LIN {X 0,Y 107.269,Z 742.199,A -85,B 0,C 180,E1 875.975,E2 875.975} C_VEL
LIN {X 0,Y 129.39,Z 733.154,A -85,B 0,C 180,E1 878.002,E2 878.002} C_VEL
LIN {X 0,Y 146.555,Z 724.699,A -85,B 0,C 180,E1 879.159,E2 879.159} C_VEL
LIN {X 0,Y 162.746,Z 715.447,A -85,B 0,C 180,E1 880.032,E2 880.032} C_VEL
LIN {X 0,Y 179.966,Z 704.09,A -85,B 0,C 180,E1 880.803,E2 880.803} C_VEL
LIN {X 0,Y 199.227,Z 689.157,A -85,B 0,C 180,E1 881.52,E2 881.52} C_VEL
LIN {X 0,Y 214.939,Z 674.846,A -85,B 0,C 180,E1 882.026,E2 882.026} C_VEL
LIN {X 0,Y 228.622,Z 660.568,A -85,B 0,C 180,E1 882.421,E2 882.421} C_VEL
LIN {X 0,Y 242.806,Z 643.596,A -85,B 0,C 180,E1 882.797,E2 882.797} C_VEL
LIN {X 0,Y 256.474,Z 624.136,A -85,B 0,C 180,E1 883.132,E2 883.132} C_VEL
LIN {X 0,Y 266.594,Z 607.239,A -85,B 0,C 180,E1 883.365,E2 883.365} C_VEL
LIN {X 0,Y 268.332,Z 604.12,A -85,B 0,C 180,E1 883.387,E2 883.387} C_VEL
LIN {X 0,Y 270.409,Z 616.789,A -85,B 0,C 180,E1 877.384,E2 877.384} C_VEL
LIN {X 0,Y 277.899,Z 632.412,A -85,B 0,C 180,E1 869.296,E2 869.296} C_VEL
LIN {X 0,Y 291.885,Z 647.885,A -85,B 0,C 180,E1 860.926,E2 860.926} C_VEL
LIN {X 0,Y 310.289,Z 661.965,A -85,B 0,C 180,E1 853.527,E2 853.527} C_VEL
LIN {X 0,Y 318.229,Z 667.453,A -85,B 0,C 180,E1 850.836,E2 850.836} C_VEL
LIN {X 0,Y 321.012,Z 670.575,A -85,B 0,C 180,E1 849.658,E2 849.658} C_VEL
LIN {X 0,Y 325.728,Z 680.817,A -85,B 0,C 180,E1 846.455,E2 846.455} C_VEL
LIN {X 0,Y 328.331,Z 683.324,A -85,B 0,C 180,E1 845.473,E2 845.473} C_VEL
LIN {X 0,Y 341.914,Z 693.088,A -85,B 0,C 180,E1 841.359,E2 841.359} C_VEL
LIN {X 0,Y 349.014,Z 698.348,A -85,B 0,C 180,E1 839.097,E2 839.097} C_VEL
LIN {X 0,Y 357.736,Z 704.336,A -85,B 0,C 180,E1 836.203,E2 836.203} C_VEL
LIN {X 0,Y 364.953,Z 709.797,A -85,B 0,C 180,E1 833.389,E2 833.389} C_VEL
LIN {X 0,Y 371.95,Z 714.302,A -85,B 0,C 180,E1 830.617,E2 830.617} C_VEL
LIN {X 0,Y 378.032,Z 719.013,A -85,B 0,C 180,E1 827.547,E2 827.547} C_VEL
LIN {X 0,Y 383.966,Z 722.788,A -85,B 0,C 180,E1 824.321,E2 824.321} C_VEL
LIN {X 0,Y 387.978,Z 724.966,A -85,B 0,C 180,E1 821.897,E2 821.897} C_VEL
LIN {X 0,Y 390.844,Z 727.557,A -85,B 0,C 180,E1 818.977,E2 818.977} C_VEL
LIN {X 0,Y 393.194,Z 729.407,A -85,B 0,C 180,E1 815.984,E2 815.984} C_VEL
LIN {X 0,Y 394.59,Z 730.377,A -85,B 0,C 180,E1 813.243,E2 813.243} C_VEL
LIN {X 0,Y 395.184,Z 730.747,A -85,B 0,C 180,E1 810.87,E2 810.87} C_VEL
LIN {X 0,Y 395.046,Z 730.672,A -85,B 0,C 180,E1 808.115,E2 808.115} C_VEL
LIN {X 0,Y 394.002,Z 729.978,A -85,B 0,C 180,E1 805.343,E2 805.343} C_VEL
LIN {X 0,Y 392.097,Z 728.62,A -85,B 0,C 180,E1 802.528,E2 802.528} C_VEL
LIN {X 0,Y 389.452,Z 726.333,A -85,B 0,C 180,E1 799.524,E2 799.524} C_VEL
LIN {X 0,Y 387.121,Z 724.477,A -85,B 0,C 180,E1 797.51,E2 797.51} C_VEL
LIN {X 0,Y 382.147,Z 721.712,A -85,B 0,C 180,E1 794.679,E2 794.679} C_VEL
LIN {X 0,Y 376.678,Z 718.012,A -85,B 0,C 180,E1 791.749,E2 791.749} C_VEL
LIN {X 0,Y 371.327,Z 713.949,A -85,B 0,C 180,E1 789.129,E2 789.129} C_VEL
LIN {X 0,Y 362.843,Z 708.32,A -85,B 0,C 180,E1 785.761,E2 785.761} C_VEL
LIN {X 0,Y 356.642,Z 703.665,A -85,B 0,C 180,E1 783.426,E2 783.426} C_VEL
LIN {X 0,Y 347.407,Z 697.149,A -85,B 0,C 180,E1 780.366,E2 780.366} C_VEL
LIN {X 0,Y 340.783,Z 692.302,A -85,B 0,C 180,E1 778.309,E2 778.309} C_VEL
LIN {X 0,Y 328.099,Z 683.168,A -85,B 0,C 180,E1 774.458,E2 774.458} C_VEL
LIN {X 0,Y 316.296,Z 675.203,A -85,B 0,C 180,E1 770.761,E2 770.761} C_VEL
LIN {X 0,Y 303.12,Z 666.365,A -85,B 0,C 180,E1 766.254,E2 766.254} C_VEL
LIN {X 0,Y 286.344,Z 653.635,A -85,B 0,C 180,E1 759.186,E2 759.186} C_VEL
LIN {X 0,Y 271.956,Z 637.387,A -85,B 0,C 180,E1 750.002,E2 750.002} C_VEL
LIN {X 0,Y 265.416,Z 622.283,A -85,B 0,C 180,E1 741.898,E2 741.898} C_VEL
LIN {X 0,Y 264.287,Z 615.394,A -85,B 0,C 180,E1 738.416,E2 738.416} C_VEL
LIN {X 0,Y 252.372,Z 633.696,A -85,B 0,C 180,E1 738.777,E2 738.777} C_VEL
LIN {X 0,Y 240.274,Z 649.718,A -85,B 0,C 180,E1 739.175,E2 739.175} C_VEL
LIN {X 0,Y 225.446,Z 666.763,A -85,B 0,C 180,E1 739.699,E2 739.699} C_VEL
LIN {X 0,Y 209.007,Z 682.763,A -85,B 0,C 180,E1 740.358,E2 740.358} C_VEL
LIN {X 0,Y 193.884,Z 695.531,A -85,B 0,C 180,E1 741.042,E2 741.042} C_VEL
LIN {X 0,Y 177.771,Z 707.42,A -85,B 0,C 180,E1 741.886,E2 741.886} C_VEL
LIN {X 0,Y 158.675,Z 719.583,A -85,B 0,C 180,E1 743.09,E2 743.09} C_VEL
LIN {X 0,Y 138.651,Z 730.166,A -85,B 0,C 180,E1 744.697,E2 744.697} C_VEL
LIN {X 0,Y 120.58,Z 738.18,A -85,B 0,C 180,E1 746.602,E2 746.602} C_VEL
LIN {X 0,Y 102.993,Z 744.699,A -85,B 0,C 180,E1 749.117,E2 749.117} C_VEL
LIN {X 0,Y 83.628,Z 750.551,A -85,B 0,C 180,E1 753.193,E2 753.193} C_VEL
LIN {X 0,Y 61.404,Z 755.521,A -85,B 0,C 180,E1 761.501,E2 761.501} C_VEL
LIN {X 0,Y 44.937,Z 758.069,A -85,B 0,C 180,E1 774.659,E2 774.659} C_VEL
LIN {X 0,Y 34.342,Z 759.187,A -85,B 0,C 180,E1 796.533,E2 796.533} C_VEL
LIN {X 0,Y 32.202,Z 759.428,A -85,B 0,C 180,E1 810,E2 810} C_VEL
LIN {X 0,Y 42.094,Z 758.434,A -85,B 0,C 180,E1 841.501,E2 841.501} C_VEL
LIN {X 0,Y 57.032,Z 756.272,A -85,B 0,C 180,E1 855.949,E2 855.949} C_VEL
LIN {X 0,Y 74.181,Z 752.843,A -85,B 0,C 180,E1 863.963,E2 863.963} C_VEL
LIN {X 0,Y 93.483,Z 747.771,A -85,B 0,C 180,E1 869.109,E2 869.109} C_VEL
LIN {X 0,Y 116.033,Z 740.018,A -85,B 0,C 180,E1 872.825,E2 872.825} C_VEL
LIN {X 0,Y 134.66,Z 732.041,A -85,B 0,C 180,E1 874.926,E2 874.926} C_VEL
LIN {X 0,Y 151.656,Z 723.44,A -85,B 0,C 180,E1 876.394,E2 876.394} C_VEL
LIN {X 0,Y 169.723,Z 712.798,A -85,B 0,C 180,E1 877.639,E2 877.639} C_VEL
LIN {X 0,Y 189.853,Z 698.694,A -85,B 0,C 180,E1 878.76,E2 878.76} C_VEL
LIN {X 0,Y 205.452,Z 685.898,A -85,B 0,C 180,E1 879.488,E2 879.488} C_VEL
LIN {X 0,Y 220.095,Z 672.179,A -85,B 0,C 180,E1 880.097,E2 880.097} C_VEL
LIN {X 0,Y 235.61,Z 655.449,A -85,B 0,C 180,E1 880.669,E2 880.669} C_VEL
LIN {X 0,Y 249.851,Z 637.246,A -85,B 0,C 180,E1 881.144,E2 881.144} C_VEL
LIN {X 0,Y 260.942,Z 620.743,A -85,B 0,C 180,E1 881.487,E2 881.487} C_VEL
LIN {X 0,Y 264.287,Z 615.394,A -85,B 0,C 180,E1 881.584,E2 881.584} C_VEL
LIN {X 0,Y 268.52,Z 631.063,A -85,B 0,C 180,E1 873.459,E2 873.459} C_VEL
LIN {X 0,Y 279.113,Z 646.63,A -85,B 0,C 180,E1 864.777,E2 864.777} C_VEL
LIN {X 0,Y 297.074,Z 661.963,A -85,B 0,C 180,E1 856.104,E2 856.104} C_VEL
LIN {X 0,Y 312.365,Z 672.625,A -85,B 0,C 180,E1 850.521,E2 850.521} C_VEL
LIN {X 0,Y 322.908,Z 679.669,A -85,B 0,C 180,E1 847.138,E2 847.138} C_VEL
LIN {X 0,Y 328.331,Z 683.324,A -85,B 0,C 180,E1 845.473,E2 845.473} C_VEL
LIN {X 0,Y 331.211,Z 686.398,A -85,B 0,C 180,E1 844.339,E2 844.339} C_VEL
LIN {X 0,Y 333.895,Z 692.764,A -85,B 0,C 180,E1 842.353,E2 842.353} C_VEL
LIN {X 0,Y 336.631,Z 697.683,A -85,B 0,C 180,E1 840.7,E2 840.7} C_VEL
LIN {X 0,Y 337.945,Z 698.909,A -85,B 0,C 180,E1 840.22,E2 840.22} C_VEL
LIN {X 0,Y 347.638,Z 706.073,A -85,B 0,C 180,E1 837.025,E2 837.025} C_VEL
LIN {X 0,Y 353.224,Z 709.991,A -85,B 0,C 180,E1 835.063,E2 835.063} C_VEL
LIN {X 0,Y 361.68,Z 716.034,A -85,B 0,C 180,E1 831.736,E2 831.736} C_VEL
LIN {X 0,Y 366.452,Z 719.165,A -85,B 0,C 180,E1 829.719,E2 829.719} C_VEL
LIN {X 0,Y 371.607,Z 723.088,A -85,B 0,C 180,E1 827.053,E2 827.053} C_VEL
LIN {X 0,Y 377.322,Z 726.693,A -85,B 0,C 180,E1 823.952,E2 823.952} C_VEL
LIN {X 0,Y 381.009,Z 728.704,A -85,B 0,C 180,E1 821.657,E2 821.657} C_VEL
LIN {X 0,Y 383.905,Z 731.334,A -85,B 0,C 180,E1 818.687,E2 818.687} C_VEL
LIN {X 0,Y 386.121,Z 733.014,A -85,B 0,C 180,E1 815.796,E2 815.796} C_VEL
LIN {X 0,Y 387.381,Z 733.865,A -85,B 0,C 180,E1 813.255,E2 813.255} C_VEL
LIN {X 0,Y 388.009,Z 734.247,A -85,B 0,C 180,E1 810.738,E2 810.738} C_VEL
LIN {X 0,Y 387.769,Z 734.088,A -85,B 0,C 180,E1 807.784,E2 807.784} C_VEL
LIN {X 0,Y 386.505,Z 733.267,A -85,B 0,C 180,E1 804.806,E2 804.806} C_VEL
LIN {X 0,Y 384.428,Z 731.79,A -85,B 0,C 180,E1 801.927,E2 801.927} C_VEL
LIN {X 0,Y 381.824,Z 729.482,A -85,B 0,C 180,E1 799.12,E2 799.12} C_VEL
LIN {X 0,Y 379.852,Z 728.001,A -85,B 0,C 180,E1 797.536,E2 797.536} C_VEL
LIN {X 0,Y 374.853,Z 725.234,A -85,B 0,C 180,E1 794.69,E2 794.69} C_VEL
LIN {X 0,Y 368.445,Z 720.785,A -85,B 0,C 180,E1 791.285,E2 791.285} C_VEL
LIN {X 0,Y 364.166,Z 717.56,A -85,B 0,C 180,E1 789.259,E2 789.259} C_VEL
LIN {X 0,Y 356.871,Z 712.735,A -85,B 0,C 180,E1 786.377,E2 786.377} C_VEL
LIN {X 0,Y 350.023,Z 707.643,A -85,B 0,C 180,E1 783.765,E2 783.765} C_VEL
LIN {X 0,Y 340.584,Z 700.983,A -85,B 0,C 180,E1 780.645,E2 780.645} C_VEL
LIN {X 0,Y 333.927,Z 696.156,A -85,B 0,C 180,E1 778.582,E2 778.582} C_VEL
LIN {X 0,Y 321.808,Z 687.707,A -85,B 0,C 180,E1 774.803,E2 774.803} C_VEL
LIN {X 0,Y 309.478,Z 679.635,A -85,B 0,C 180,E1 770.843,E2 770.843} C_VEL
LIN {X 0,Y 295.929,Z 670.716,A -85,B 0,C 180,E1 766.029,E2 766.029} C_VEL
LIN {X 0,Y 276.611,Z 655.55,A -85,B 0,C 180,E1 757.133,E2 757.133} C_VEL
LIN {X 0,Y 264.634,Z 639.785,A -85,B 0,C 180,E1 747.869,E2 747.869} C_VEL
LIN {X 0,Y 260.096,Z 626.207,A -85,B 0,C 180,E1 740.301,E2 740.301} C_VEL
LIN {X 0,Y 246.055,Z 645.77,A -85,B 0,C 180,E1 740.85,E2 740.85} C_VEL
LIN {X 0,Y 233.011,Z 661.342,A -85,B 0,C 180,E1 741.4,E2 741.4} C_VEL
LIN {X 0,Y 217.846,Z 677.117,A -85,B 0,C 180,E1 742.109,E2 742.109} C_VEL
LIN {X 0,Y 198.945,Z 693.776,A -85,B 0,C 180,E1 743.129,E2 743.129} C_VEL
LIN {X 0,Y 182.954,Z 705.845,A -85,B 0,C 180,E1 744.137,E2 744.137} C_VEL
LIN {X 0,Y 167.013,Z 716.333,A -85,B 0,C 180,E1 745.325,E2 745.325} C_VEL
LIN {X 0,Y 148.173,Z 727.054,A -85,B 0,C 180,E1 747.047,E2 747.047} C_VEL
LIN {X 0,Y 127.535,Z 736.741,A -85,B 0,C 180,E1 749.526,E2 749.526} C_VEL
LIN {X 0,Y 109.127,Z 743.853,A -85,B 0,C 180,E1 752.559,E2 752.559} C_VEL
LIN {X 0,Y 92.082,Z 749.289,A -85,B 0,C 180,E1 756.541,E2 756.541} C_VEL
LIN {X 0,Y 73.08,Z 754.138,A -85,B 0,C 180,E1 763.527,E2 763.527} C_VEL
LIN {X 0,Y 53.864,Z 757.62,A -85,B 0,C 180,E1 777.435,E2 777.435} C_VEL
LIN {X 0,Y 43.024,Z 758.946,A -85,B 0,C 180,E1 796.563,E2 796.563} C_VEL
LIN {X 0,Y 40.271,Z 759.252,A -85,B 0,C 180,E1 810,E2 810} C_VEL
LIN {X 0,Y 49.221,Z 758.259,A -85,B 0,C 180,E1 836.542,E2 836.542} C_VEL
LIN {X 0,Y 62.984,Z 756.097,A -85,B 0,C 180,E1 850.602,E2 850.602} C_VEL
LIN {X 0,Y 79.267,Z 752.667,A -85,B 0,C 180,E1 859.178,E2 859.178} C_VEL
LIN {X 0,Y 97.707,Z 747.66,A -85,B 0,C 180,E1 864.942,E2 864.942} C_VEL
LIN {X 0,Y 119.744,Z 739.942,A -85,B 0,C 180,E1 869.312,E2 869.312} C_VEL
LIN {X 0,Y 138.318,Z 731.866,A -85,B 0,C 180,E1 871.862,E2 871.862} C_VEL
LIN {X 0,Y 155.589,Z 722.999,A -85,B 0,C 180,E1 873.677,E2 873.677} C_VEL
LIN {X 0,Y 174.976,Z 711.371,A -85,B 0,C 180,E1 875.295,E2 875.295} C_VEL
LIN {X 0,Y 193.946,Z 697.729,A -85,B 0,C 180,E1 876.571,E2 876.571} C_VEL
LIN {X 0,Y 208.96,Z 685.255,A -85,B 0,C 180,E1 877.427,E2 877.427} C_VEL
LIN {X 0,Y 223.985,Z 671.009,A -85,B 0,C 180,E1 878.188,E2 878.188} C_VEL
LIN {X 0,Y 240.536,Z 652.677,A -85,B 0,C 180,E1 878.924,E2 878.924} C_VEL
LIN {X 0,Y 253.48,Z 635.791,A -85,B 0,C 180,E1 879.447,E2 879.447} C_VEL
LIN {X 0,Y 260.141,Z 626.204,A -85,B 0,C 180,E1 879.672,E2 879.672} C_VEL
LIN {X 0,Y 266.173,Z 642.618,A -85,B 0,C 180,E1 870.521,E2 870.521} C_VEL
LIN {X 0,Y 279.562,Z 658.292,A -85,B 0,C 180,E1 861.224,E2 861.224} C_VEL
LIN {X 0,Y 297.375,Z 671.692,A -85,B 0,C 180,E1 853.425,E2 853.425} C_VEL
LIN {X 0,Y 313.212,Z 681.934,A -85,B 0,C 180,E1 847.953,E2 847.953} C_VEL
LIN {X 0,Y 326.167,Z 690.696,A -85,B 0,C 180,E1 843.822,E2 843.822} C_VEL
LIN {X 0,Y 337.945,Z 698.909,A -85,B 0,C 180,E1 840.22,E2 840.22} C_VEL
LIN {X 0,Y 340.504,Z 701.924,A -85,B 0,C 180,E1 839.093,E2 839.093} C_VEL
LIN {X 0,Y 342.63,Z 707.797,A -85,B 0,C 180,E1 837.094,E2 837.094} C_VEL
LIN {X 0,Y 344.798,Z 712.184,A -85,B 0,C 180,E1 835.411,E2 835.411} C_VEL
LIN {X 0,Y 345.911,Z 713.261,A -85,B 0,C 180,E1 834.918,E2 834.918} C_VEL
LIN {X 0,Y 353.809,Z 718.973,A -85,B 0,C 180,E1 831.813,E2 831.813} C_VEL
LIN {X 0,Y 359.008,Z 722.341,A -85,B 0,C 180,E1 829.692,E2 829.692} C_VEL
LIN {X 0,Y 365.746,Z 727.384,A -85,B 0,C 180,E1 826.189,E2 826.189} C_VEL
LIN {X 0,Y 371.491,Z 730.767,A -85,B 0,C 180,E1 823.005,E2 823.005} C_VEL
LIN {X 0,Y 373.946,Z 732.244,A -85,B 0,C 180,E1 821.411,E2 821.411} C_VEL
LIN {X 0,Y 376.54,Z 734.529,A -85,B 0,C 180,E1 818.705,E2 818.705} C_VEL
LIN {X 0,Y 378.892,Z 736.29,A -85,B 0,C 180,E1 815.603,E2 815.603} C_VEL
LIN {X 0,Y 380.159,Z 737.174,A -85,B 0,C 180,E1 813.015,E2 813.015} C_VEL
LIN {X 0,Y 380.798,Z 737.533,A -85,B 0,C 180,E1 810.15,E2 810.15} C_VEL
LIN {X 0,Y 380.314,Z 737.257,A -85,B 0,C 180,E1 807.288,E2 807.288} C_VEL
LIN {X 0,Y 378.913,Z 736.322,A -85,B 0,C 180,E1 804.398,E2 804.398} C_VEL
LIN {X 0,Y 376.557,Z 734.557,A -85,B 0,C 180,E1 801.296,E2 801.296} C_VEL
LIN {X 0,Y 373.944,Z 732.241,A -85,B 0,C 180,E1 798.589,E2 798.589} C_VEL
LIN {X 0,Y 370.394,Z 730.171,A -85,B 0,C 180,E1 796.369,E2 796.369} C_VEL
LIN {X 0,Y 364.724,Z 726.669,A -85,B 0,C 180,E1 793.273,E2 793.273} C_VEL
LIN {X 0,Y 358.487,Z 721.913,A -85,B 0,C 180,E1 790.045,E2 790.045} C_VEL
LIN {X 0,Y 350.002,Z 716.376,A -85,B 0,C 180,E1 786.683,E2 786.683} C_VEL
LIN {X 0,Y 343.175,Z 711.297,A -85,B 0,C 180,E1 784.088,E2 784.088} C_VEL
LIN {X 0,Y 333.8,Z 704.65,A -85,B 0,C 180,E1 781.007,E2 781.007} C_VEL
LIN {X 0,Y 327.053,Z 699.942,A -85,B 0,C 180,E1 778.875,E2 778.875} C_VEL
LIN {X 0,Y 315.457,Z 692.098,A -85,B 0,C 180,E1 775.179,E2 775.179} C_VEL
LIN {X 0,Y 303.645,Z 684.586,A -85,B 0,C 180,E1 771.3,E2 771.3} C_VEL
LIN {X 0,Y 290.349,Z 676.086,A -85,B 0,C 180,E1 766.476,E2 766.476} C_VEL
LIN {X 0,Y 272.311,Z 662.492,A -85,B 0,C 180,E1 758.088,E2 758.088} C_VEL
LIN {X 0,Y 260.475,Z 648.09,A -85,B 0,C 180,E1 749.178,E2 749.178} C_VEL
LIN {X 0,Y 255.921,Z 636.352,A -85,B 0,C 180,E1 742.271,E2 742.271} C_VEL
LIN {X 0,Y 241.56,Z 654.96,A -85,B 0,C 180,E1 742.947,E2 742.947} C_VEL
LIN {X 0,Y 226.121,Z 671.834,A -85,B 0,C 180,E1 743.764,E2 743.764} C_VEL
LIN {X 0,Y 212.205,Z 685.081,A -85,B 0,C 180,E1 744.595,E2 744.595} C_VEL
LIN {X 0,Y 197.315,Z 697.555,A -85,B 0,C 180,E1 745.593,E2 745.593} C_VEL
LIN {X 0,Y 178.532,Z 711.192,A -85,B 0,C 180,E1 747.079,E2 747.079} C_VEL
LIN {X 0,Y 159.871,Z 722.548,A -85,B 0,C 180,E1 748.897,E2 748.897} C_VEL
LIN {X 0,Y 143.318,Z 731.222,A -85,B 0,C 180,E1 750.905,E2 750.905} C_VEL
LIN {X 0,Y 125.066,Z 739.366,A -85,B 0,C 180,E1 753.762,E2 753.762} C_VEL
LIN {X 0,Y 103.54,Z 747.206,A -85,B 0,C 180,E1 758.545,E2 758.545} C_VEL
LIN {X 0,Y 85.7,Z 752.281,A -85,B 0,C 180,E1 764.634,E2 764.634} C_VEL
LIN {X 0,Y 70.152,Z 755.771,A -85,B 0,C 180,E1 773.234,E2 773.234} C_VEL
LIN {X 0,Y 57.199,Z 757.992,A -85,B 0,C 180,E1 786.296,E2 786.296} C_VEL
LIN {X 0,Y 48.688,Z 759.027,A -85,B 0,C 180,E1 807.646,E2 807.646} C_VEL
LIN {X 0,Y 48.507,Z 759.055,A -85,B 0,C 180,E1 811.181,E2 811.181} C_VEL
LIN {X 0,Y 56.626,Z 758.083,A -85,B 0,C 180,E1 832.856,E2 832.856} C_VEL
LIN {X 0,Y 69.404,Z 755.919,A -85,B 0,C 180,E1 846.218,E2 846.218} C_VEL
LIN {X 0,Y 84.84,Z 752.491,A -85,B 0,C 180,E1 854.995,E2 854.995} C_VEL
LIN {X 0,Y 102.624,Z 747.483,A -85,B 0,C 180,E1 861.201,E2 861.201} C_VEL
LIN {X 0,Y 124.115,Z 739.766,A -85,B 0,C 180,E1 866.065,E2 866.065} C_VEL
LIN {X 0,Y 142.35,Z 731.691,A -85,B 0,C 180,E1 868.963,E2 868.963} C_VEL
LIN {X 0,Y 158.893,Z 723.089,A -85,B 0,C 180,E1 870.996,E2 870.996} C_VEL
LIN {X 0,Y 177.546,Z 711.828,A -85,B 0,C 180,E1 872.835,E2 872.835} C_VEL
LIN {X 0,Y 196.325,Z 698.346,A -85,B 0,C 180,E1 874.335,E2 874.335} C_VEL
LIN {X 0,Y 211.211,Z 685.969,A -85,B 0,C 180,E1 875.343,E2 875.343} C_VEL
LIN {X 0,Y 225.472,Z 672.485,A -85,B 0,C 180,E1 876.199,E2 876.199} C_VEL
LIN {X 0,Y 240.066,Z 656.668,A -85,B 0,C 180,E1 876.978,E2 876.978} C_VEL
LIN {X 0,Y 255.02,Z 637.615,A -85,B 0,C 180,E1 877.697,E2 877.697} C_VEL
LIN {X 0,Y 255.92,Z 636.353,A -85,B 0,C 180,E1 877.729,E2 877.729} C_VEL
LIN {X 0,Y 261.843,Z 650.287,A -85,B 0,C 180,E1 869.477,E2 869.477} C_VEL
LIN {X 0,Y 275.337,Z 665.068,A -85,B 0,C 180,E1 860.272,E2 860.272} C_VEL
LIN {X 0,Y 293.517,Z 678.123,A -85,B 0,C 180,E1 852.334,E2 852.334} C_VEL
LIN {X 0,Y 308.965,Z 687.933,A -85,B 0,C 180,E1 846.931,E2 846.931} C_VEL
LIN {X 0,Y 320.012,Z 695.161,A -85,B 0,C 180,E1 843.356,E2 843.356} C_VEL
LIN {X 0,Y 332.15,Z 703.395,A -85,B 0,C 180,E1 839.542,E2 839.542} C_VEL
LIN {X 0,Y 342.207,Z 710.655,A -85,B 0,C 180,E1 836.231,E2 836.231} C_VEL
LIN {X 0,Y 345.911,Z 713.261,A -85,B 0,C 180,E1 834.918,E2 834.918} C_VEL
LIN {X 0,Y 348.008,Z 715.895,A -85,B 0,C 180,E1 833.766,E2 833.766} C_VEL
LIN {X 0,Y 349.396,Z 720.843,A -85,B 0,C 180,E1 831.73,E2 831.73} C_VEL
LIN {X 0,Y 350.965,Z 724.671,A -85,B 0,C 180,E1 829.923,E2 829.923} C_VEL
LIN {X 0,Y 351.697,Z 725.376,A -85,B 0,C 180,E1 829.498,E2 829.498} C_VEL
LIN {X 0,Y 357.601,Z 729.875,A -85,B 0,C 180,E1 826.45,E2 826.45} C_VEL
LIN {X 0,Y 363.57,Z 733.555,A -85,B 0,C 180,E1 823.193,E2 823.193} C_VEL
LIN {X 0,Y 366.547,Z 735.242,A -85,B 0,C 180,E1 821.325,E2 821.325} C_VEL
LIN {X 0,Y 369.316,Z 737.667,A -85,B 0,C 180,E1 818.406,E2 818.406} C_VEL
LIN {X 0,Y 371.477,Z 739.292,A -85,B 0,C 180,E1 815.56,E2 815.56} C_VEL
LIN {X 0,Y 372.784,Z 740.227,A -85,B 0,C 180,E1 812.921,E2 812.921} C_VEL
LIN {X 0,Y 373.392,Z 740.56,A -85,B 0,C 180,E1 810.153,E2 810.153} C_VEL
LIN {X 0,Y 372.937,Z 740.298,A -85,B 0,C 180,E1 807.388,E2 807.388} C_VEL
LIN {X 0,Y 371.597,Z 739.388,A -85,B 0,C 180,E1 804.597,E2 804.597} C_VEL
LIN {X 0,Y 369.19,Z 737.558,A -85,B 0,C 180,E1 801.435,E2 801.435} C_VEL
LIN {X 0,Y 366.342,Z 735.039,A -85,B 0,C 180,E1 798.48,E2 798.48} C_VEL
LIN {X 0,Y 361.897,Z 732.59,A -85,B 0,C 180,E1 795.88,E2 795.88} C_VEL
LIN {X 0,Y 355.961,Z 728.726,A -85,B 0,C 180,E1 792.68,E2 792.68} C_VEL
LIN {X 0,Y 350.526,Z 724.613,A -85,B 0,C 180,E1 789.986,E2 789.986} C_VEL
LIN {X 0,Y 342.413,Z 719.253,A -85,B 0,C 180,E1 786.786,E2 786.786} C_VEL
LIN {X 0,Y 336.014,Z 714.519,A -85,B 0,C 180,E1 784.376,E2 784.376} C_VEL
LIN {X 0,Y 324.126,Z 706.096,A -85,B 0,C 180,E1 780.428,E2 780.428} C_VEL
LIN {X 0,Y 309.625,Z 696.7,A -85,B 0,C 180,E1 775.763,E2 775.763} C_VEL
LIN {X 0,Y 297.231,Z 689.097,A -85,B 0,C 180,E1 771.612,E2 771.612} C_VEL
LIN {X 0,Y 283.693,Z 680.67,A -85,B 0,C 180,E1 766.557,E2 766.557} C_VEL
LIN {X 0,Y 264.087,Z 665.609,A -85,B 0,C 180,E1 756.743,E2 756.743} C_VEL
LIN {X 0,Y 253.303,Z 650.505,A -85,B 0,C 180,E1 746.998,E2 746.998} C_VEL
LIN {X 0,Y 251.509,Z 646.37,A -85,B 0,C 180,E1 744.318,E2 744.318} C_VEL
LIN {X 0,Y 238.889,Z 661.556,A -85,B 0,C 180,E1 745.034,E2 745.034} C_VEL
LIN {X 0,Y 223.467,Z 677.724,A -85,B 0,C 180,E1 746.008,E2 746.008} C_VEL
LIN {X 0,Y 205.863,Z 693.428,A -85,B 0,C 180,E1 747.287,E2 747.287} C_VEL
LIN {X 0,Y 189.786,Z 705.782,A -85,B 0,C 180,E1 748.649,E2 748.649} C_VEL
LIN {X 0,Y 172.662,Z 717.219,A -85,B 0,C 180,E1 750.374,E2 750.374} C_VEL
LIN {X 0,Y 151.486,Z 729.173,A -85,B 0,C 180,E1 753.055,E2 753.055} C_VEL
LIN {X 0,Y 133.52,Z 737.59,A -85,B 0,C 180,E1 756.034,E2 756.034} C_VEL
LIN {X 0,Y 116.912,Z 744.168,A -85,B 0,C 180,E1 759.68,E2 759.68} C_VEL
LIN {X 0,Y 99.21,Z 750.021,A -85,B 0,C 180,E1 765.139,E2 765.139} C_VEL
LIN {X 0,Y 79.791,Z 754.994,A -85,B 0,C 180,E1 774.805,E2 774.805} C_VEL
LIN {X 0,Y 66.07,Z 757.597,A -85,B 0,C 180,E1 787.393,E2 787.393} C_VEL
LIN {X 0,Y 57.987,Z 758.692,A -85,B 0,C 180,E1 803.068,E2 803.068} C_VEL
LIN {X 0,Y 56.435,Z 758.898,A -85,B 0,C 180,E1 810,E2 810} C_VEL
LIN {X 0,Y 64.212,Z 757.908,A -85,B 0,C 180,E1 830.031,E2 830.031} C_VEL
LIN {X 0,Y 76.854,Z 755.595,A -85,B 0,C 180,E1 843.117,E2 843.117} C_VEL
LIN {X 0,Y 92.458,Z 751.895,A -85,B 0,C 180,E1 852.099,E2 852.099} C_VEL
LIN {X 0,Y 112.396,Z 745.831,A -85,B 0,C 180,E1 859.119,E2 859.119} C_VEL
LIN {X 0,Y 131.131,Z 738.613,A -85,B 0,C 180,E1 863.505,E2 863.505} C_VEL
LIN {X 0,Y 148.64,Z 730.573,A -85,B 0,C 180,E1 866.523,E2 866.523} C_VEL
LIN {X 0,Y 167.824,Z 720.187,A -85,B 0,C 180,E1 869.074,E2 869.074} C_VEL
LIN {X 0,Y 187.254,Z 707.599,A -85,B 0,C 180,E1 871.116,E2 871.116} C_VEL
LIN {X 0,Y 203.993,Z 694.934,A -85,B 0,C 180,E1 872.565,E2 872.565} C_VEL
LIN {X 0,Y 220.623,Z 680.462,A -85,B 0,C 180,E1 873.797,E2 873.797} C_VEL
LIN {X 0,Y 236.75,Z 663.978,A -85,B 0,C 180,E1 874.837,E2 874.837} C_VEL
LIN {X 0,Y 249.778,Z 648.572,A -85,B 0,C 180,E1 875.586,E2 875.586} C_VEL
LIN {X 0,Y 251.641,Z 646.265,A -85,B 0,C 180,E1 875.66,E2 875.66} C_VEL
LIN {X 0,Y 259.189,Z 660.243,A -85,B 0,C 180,E1 866.783,E2 866.783} C_VEL
LIN {X 0,Y 275.131,Z 674.81,A -85,B 0,C 180,E1 857.187,E2 857.187} C_VEL
LIN {X 0,Y 292.585,Z 686.266,A -85,B 0,C 180,E1 850.048,E2 850.048} C_VEL
LIN {X 0,Y 304.152,Z 693.366,A -85,B 0,C 180,E1 846.029,E2 846.029} C_VEL
LIN {X 0,Y 313.449,Z 699.205,A -85,B 0,C 180,E1 842.969,E2 842.969} C_VEL
LIN {X 0,Y 325.836,Z 707.364,A -85,B 0,C 180,E1 838.999,E2 838.999} C_VEL
LIN {X 0,Y 337.159,Z 715.236,A -85,B 0,C 180,E1 835.241,E2 835.241} C_VEL
LIN {X 0,Y 345.295,Z 721.29,A -85,B 0,C 180,E1 832.082,E2 832.082} C_VEL
LIN {X 0,Y 351.697,Z 725.376,A -85,B 0,C 180,E1 829.498,E2 829.498} C_VEL
LIN {X 0,Y 353.067,Z 727.575,A -85,B 0,C 180,E1 828.308,E2 828.308} C_VEL
LIN {X 0,Y 353.045,Z 732.334,A -85,B 0,C 180,E1 825.975,E2 825.975} C_VEL
LIN {X 0,Y 353.795,Z 734.902,A -85,B 0,C 180,E1 824.398,E2 824.398} C_VEL
LIN {X 0,Y 354.44,Z 735.401,A -85,B 0,C 180,E1 823.965,E2 823.965} C_VEL
LIN {X 0,Y 359.026,Z 737.928,A -85,B 0,C 180,E1 821.24,E2 821.24} C_VEL
LIN {X 0,Y 361.876,Z 740.472,A -85,B 0,C 180,E1 818.26,E2 818.26} C_VEL
LIN {X 0,Y 363.94,Z 741.973,A -85,B 0,C 180,E1 815.517,E2 815.517} C_VEL
LIN {X 0,Y 365.252,Z 742.863,A -85,B 0,C 180,E1 812.824,E2 812.824} C_VEL
LIN {X 0,Y 365.802,Z 743.157,A -85,B 0,C 180,E1 810,E2 810} C_VEL
LIN {X 0,Y 365.288,Z 742.874,A -85,B 0,C 180,E1 807.176,E2 807.176} C_VEL
LIN {X 0,Y 363.857,Z 741.936,A -85,B 0,C 180,E1 804.323,E2 804.323} C_VEL
LIN {X 0,Y 361.603,Z 740.212,A -85,B 0,C 180,E1 801.414,E2 801.414} C_VEL
LIN {X 0,Y 358.832,Z 737.738,A -85,B 0,C 180,E1 798.591,E2 798.591} C_VEL
LIN {X 0,Y 353.881,Z 735.061,A -85,B 0,C 180,E1 795.731,E2 795.731} C_VEL
LIN {X 0,Y 347.315,Z 730.61,A -85,B 0,C 180,E1 792.234,E2 792.234} C_VEL
LIN {X 0,Y 343.184,Z 727.506,A -85,B 0,C 180,E1 790.235,E2 790.235} C_VEL
LIN {X 0,Y 334.755,Z 721.871,A -85,B 0,C 180,E1 786.923,E2 786.923} C_VEL
LIN {X 0,Y 329.196,Z 717.734,A -85,B 0,C 180,E1 784.838,E2 784.838} C_VEL
LIN {X 0,Y 316.674,Z 709.251,A -85,B 0,C 180,E1 780.629,E2 780.629} C_VEL
LIN {X 0,Y 302.644,Z 700.528,A -85,B 0,C 180,E1 776.024,E2 776.024} C_VEL
LIN {X 0,Y 290.765,Z 693.49,A -85,B 0,C 180,E1 771.952,E2 771.952} C_VEL
LIN {X 0,Y 277.704,Z 685.613,A -85,B 0,C 180,E1 766.963,E2 766.963} C_VEL
LIN {X 0,Y 259.478,Z 672.257,A -85,B 0,C 180,E1 757.785,E2 757.785} C_VEL
LIN {X 0,Y 248.86,Z 658.802,A -85,B 0,C 180,E1 748.563,E2 748.563} C_VEL
LIN {X 0,Y 247.373,Z 655.693,A -85,B 0,C 180,E1 746.443,E2 746.443} C_VEL
LIN {X 0,Y 232.628,Z 671.988,A -85,B 0,C 180,E1 747.444,E2 747.444} C_VEL
LIN {X 0,Y 218.474,Z 685.621,A -85,B 0,C 180,E1 748.525,E2 748.525} C_VEL
LIN {X 0,Y 201.945,Z 699.573,A -85,B 0,C 180,E1 749.962,E2 749.962} C_VEL
LIN {X 0,Y 182.666,Z 713.333,A -85,B 0,C 180,E1 751.969,E2 751.969} C_VEL
LIN {X 0,Y 166.459,Z 723.279,A -85,B 0,C 180,E1 754.022,E2 754.022} C_VEL
LIN {X 0,Y 148.251,Z 732.934,A -85,B 0,C 180,E1 756.889,E2 756.889} C_VEL
LIN {X 0,Y 127.092,Z 742.182,A -85,B 0,C 180,E1 761.366,E2 761.366} C_VEL
LIN {X 0,Y 110.186,Z 748.215,A -85,B 0,C 180,E1 766.404,E2 766.404} C_VEL
LIN {X 0,Y 94.762,Z 752.77,A -85,B 0,C 180,E1 773.033,E2 773.033} C_VEL
LIN {X 0,Y 78.942,Z 756.508,A -85,B 0,C 180,E1 784.065,E2 784.065} C_VEL
LIN {X 0,Y 67.648,Z 758.352,A -85,B 0,C 180,E1 799.785,E2 799.785} C_VEL
LIN {X 0,Y 64.525,Z 758.721,A -85,B 0,C 180,E1 810,E2 810} C_VEL
LIN {X 0,Y 71.923,Z 757.732,A -85,B 0,C 180,E1 827.807,E2 827.807} C_VEL
LIN {X 0,Y 83.818,Z 755.42,A -85,B 0,C 180,E1 840.064,E2 840.064} C_VEL
LIN {X 0,Y 98.679,Z 751.719,A -85,B 0,C 180,E1 848.913,E2 848.913} C_VEL
LIN {X 0,Y 117.911,Z 745.653,A -85,B 0,C 180,E1 856.113,E2 856.113} C_VEL
LIN {X 0,Y 135.747,Z 738.615,A -85,B 0,C 180,E1 860.652,E2 860.652} C_VEL
LIN {X 0,Y 153.282,Z 730.403,A -85,B 0,C 180,E1 863.976,E2 863.976} C_VEL
LIN {X 0,Y 171.202,Z 720.559,A -85,B 0,C 180,E1 866.622,E2 866.622} C_VEL
LIN {X 0,Y 190.351,Z 708.126,A -85,B 0,C 180,E1 868.882,E2 868.882} C_VEL
LIN {X 0,Y 207.29,Z 695.223,A -85,B 0,C 180,E1 870.527,E2 870.527} C_VEL
LIN {X 0,Y 222.37,Z 682.065,A -85,B 0,C 180,E1 871.787,E2 871.787} C_VEL
LIN {X 0,Y 238.988,Z 665.302,A -85,B 0,C 180,E1 873.004,E2 873.004} C_VEL
LIN {X 0,Y 247.471,Z 655.599,A -85,B 0,C 180,E1 873.554,E2 873.554} C_VEL
LIN {X 0,Y 256.597,Z 669.338,A -85,B 0,C 180,E1 864.232,E2 864.232} C_VEL
LIN {X 0,Y 274.915,Z 683.771,A -85,B 0,C 180,E1 854.233,E2 854.233} C_VEL
LIN {X 0,Y 288.659,Z 692.258,A -85,B 0,C 180,E1 848.796,E2 848.796} C_VEL
LIN {X 0,Y 298.233,Z 697.916,A -85,B 0,C 180,E1 845.441,E2 845.441} C_VEL
LIN {X 0,Y 307.04,Z 703.272,A -85,B 0,C 180,E1 842.494,E2 842.494} C_VEL
LIN {X 0,Y 318.914,Z 710.736,A -85,B 0,C 180,E1 838.612,E2 838.612} C_VEL
LIN {X 0,Y 330.713,Z 718.758,A -85,B 0,C 180,E1 834.657,E2 834.657} C_VEL
LIN {X 0,Y 338.877,Z 724.758,A -85,B 0,C 180,E1 831.458,E2 831.458} C_VEL
LIN {X 0,Y 344.827,Z 728.656,A -85,B 0,C 180,E1 829.038,E2 829.038} C_VEL
LIN {X 0,Y 350.602,Z 732.943,A -85,B 0,C 180,E1 826.033,E2 826.033} C_VEL
LIN {X 0,Y 354.44,Z 735.401,A -85,B 0,C 180,E1 823.965,E2 823.965} C_VEL
LIN {X 0,Y 355.505,Z 736.832,A -85,B 0,C 180,E1 822.837,E2 822.837} C_VEL
LIN {X 0,Y 354.907,Z 739.32,A -85,B 0,C 180,E1 821.171,E2 821.171} C_VEL
LIN {X 0,Y 353.819,Z 742.122,A -85,B 0,C 180,E1 819.019,E2 819.019} C_VEL
LIN {X 0,Y 354.148,Z 742.749,A -85,B 0,C 180,E1 818.296,E2 818.296} C_VEL
LIN {X 0,Y 356.383,Z 744.365,A -85,B 0,C 180,E1 815.312,E2 815.312} C_VEL
LIN {X 0,Y 357.77,Z 745.34,A -85,B 0,C 180,E1 812.402,E2 812.402} C_VEL
LIN {X 0,Y 358.118,Z 745.51,A -85,B 0,C 180,E1 809.68,E2 809.68} C_VEL
LIN {X 0,Y 357.607,Z 745.215,A -85,B 0,C 180,E1 807.116,E2 807.116} C_VEL
LIN {X 0,Y 356.195,Z 744.256,A -85,B 0,C 180,E1 804.362,E2 804.362} C_VEL
LIN {X 0,Y 353.751,Z 742.396,A -85,B 0,C 180,E1 801.222,E2 801.222} C_VEL
LIN {X 0,Y 351.16,Z 740.172,A -85,B 0,C 180,E1 798.671,E2 798.671} C_VEL
LIN {X 0,Y 345.403,Z 736.96,A -85,B 0,C 180,E1 795.415,E2 795.415} C_VEL
LIN {X 0,Y 339.232,Z 732.666,A -85,B 0,C 180,E1 792.152,E2 792.152} C_VEL
LIN {X 0,Y 335.244,Z 729.795,A -85,B 0,C 180,E1 790.307,E2 790.307} C_VEL
LIN {X 0,Y 326.87,Z 724.064,A -85,B 0,C 180,E1 787.037,E2 787.037} C_VEL
LIN {X 0,Y 321.781,Z 720.435,A -85,B 0,C 180,E1 785.142,E2 785.142} C_VEL
LIN {X 0,Y 309.75,Z 712.6,A -85,B 0,C 180,E1 781.044,E2 781.044} C_VEL
LIN {X 0,Y 296.174,Z 704.522,A -85,B 0,C 180,E1 776.5,E2 776.5} C_VEL
LIN {X 0,Y 284.24,Z 697.739,A -85,B 0,C 180,E1 772.326,E2 772.326} C_VEL
LIN {X 0,Y 270.701,Z 689.832,A -85,B 0,C 180,E1 767,E2 767} C_VEL
LIN {X 0,Y 250.906,Z 674.917,A -85,B 0,C 180,E1 756.143,E2 756.143} C_VEL
LIN {X 0,Y 243.129,Z 664.71,A -85,B 0,C 180,E1 748.67,E2 748.67} C_VEL
LIN {X 0,Y 226.312,Z 681.891,A -85,B 0,C 180,E1 750.02,E2 750.02} C_VEL
LIN {X 0,Y 211.872,Z 694.661,A -85,B 0,C 180,E1 751.342,E2 751.342} C_VEL
LIN {X 0,Y 194.677,Z 707.953,A -85,B 0,C 180,E1 753.167,E2 753.167} C_VEL
LIN {X 0,Y 174.27,Z 721.292,A -85,B 0,C 180,E1 755.82,E2 755.82} C_VEL
LIN {X 0,Y 157.303,Z 730.697,A -85,B 0,C 180,E1 758.58,E2 758.58} C_VEL
LIN {X 0,Y 140.049,Z 738.899,A -85,B 0,C 180,E1 762.154,E2 762.154} C_VEL
LIN {X 0,Y 120.119,Z 746.753,A -85,B 0,C 180,E1 767.804,E2 767.804} C_VEL
LIN {X 0,Y 103.653,Z 751.963,A -85,B 0,C 180,E1 774.64,E2 774.64} C_VEL
LIN {X 0,Y 89.074,Z 755.695,A -85,B 0,C 180,E1 784.041,E2 784.041} C_VEL
LIN {X 0,Y 77.142,Z 758.04,A -85,B 0,C 180,E1 798.033,E2 798.033} C_VEL
LIN {X 0,Y 72.62,Z 758.545,A -85,B 0,C 180,E1 810,E2 810} C_VEL
LIN {X 0,Y 79.725,Z 757.557,A -85,B 0,C 180,E1 826.015,E2 826.015} C_VEL
LIN {X 0,Y 90.983,Z 755.244,A -85,B 0,C 180,E1 837.485,E2 837.485} C_VEL
LIN {X 0,Y 105.272,Z 751.515,A -85,B 0,C 180,E1 846.163,E2 846.163} C_VEL
LIN {X 0,Y 124.566,Z 745.145,A -85,B 0,C 180,E1 853.648,E2 853.648} C_VEL
LIN {X 0,Y 141.957,Z 738.039,A -85,B 0,C 180,E1 858.29,E2 858.29} C_VEL
LIN {X 0,Y 160.051,Z 729.291,A -85,B 0,C 180,E1 861.911,E2 861.911} C_VEL
LIN {X 0,Y 179.562,Z 718.083,A -85,B 0,C 180,E1 864.93,E2 864.93} C_VEL
LIN {X 0,Y 196.885,Z 706.326,A -85,B 0,C 180,E1 867.084,E2 867.084} C_VEL
LIN {X 0,Y 212.833,Z 693.871,A -85,B 0,C 180,E1 868.751,E2 868.751} C_VEL
LIN {X 0,Y 230.06,Z 678.328,A -85,B 0,C 180,E1 870.299,E2 870.299} C_VEL
LIN {X 0,Y 243.237,Z 664.642,A -85,B 0,C 180,E1 871.312,E2 871.312} C_VEL
LIN {X 0,Y 255.579,Z 679.301,A -85,B 0,C 180,E1 860.67,E2 860.67} C_VEL
LIN {X 0,Y 272.121,Z 690.695,A -85,B 0,C 180,E1 852.391,E2 852.391} C_VEL
LIN {X 0,Y 286.942,Z 699.182,A -85,B 0,C 180,E1 846.729,E2 846.729} C_VEL
LIN {X 0,Y 300.048,Z 706.84,A -85,B 0,C 180,E1 842.173,E2 842.173} C_VEL
LIN {X 0,Y 312.381,Z 714.314,A -85,B 0,C 180,E1 838.064,E2 838.064} C_VEL
LIN {X 0,Y 324.186,Z 722.041,A -85,B 0,C 180,E1 834.021,E2 834.021} C_VEL
LIN {X 0,Y 332.543,Z 728.085,A -85,B 0,C 180,E1 830.753,E2 830.753} C_VEL
LIN {X 0,Y 337.671,Z 731.401,A -85,B 0,C 180,E1 828.636,E2 828.636} C_VEL
LIN {X 0,Y 343.659,Z 735.831,A -85,B 0,C 180,E1 825.524,E2 825.524} C_VEL
LIN {X 0,Y 349.654,Z 739.352,A -85,B 0,C 180,E1 822.215,E2 822.215} C_VEL
LIN {X 0,Y 351.763,Z 740.672,A -85,B 0,C 180,E1 820.812,E2 820.812} C_VEL
LIN {X 0,Y 354.148,Z 742.749,A -85,B 0,C 180,E1 818.296,E2 818.296} C_VEL
LIN {X 0,Y 354.24,Z 743.775,A -85,B 0,C 180,E1 817.143,E2 817.143} C_VEL
LIN {X 0,Y 352.119,Z 745.602,A -85,B 0,C 180,E1 815.29,E2 815.29} C_VEL
LIN {X 0,Y 350.032,Z 747.097,A -85,B 0,C 180,E1 813.398,E2 813.398} C_VEL
LIN {X 0,Y 349.976,Z 747.414,A -85,B 0,C 180,E1 812.57,E2 812.57} C_VEL
LIN {X 0,Y 350.404,Z 747.634,A -85,B 0,C 180,E1 809.673,E2 809.673} C_VEL
LIN {X 0,Y 349.853,Z 747.319,A -85,B 0,C 180,E1 807.052,E2 807.052} C_VEL
LIN {X 0,Y 348.347,Z 746.259,A -85,B 0,C 180,E1 804.235,E2 804.235} C_VEL
LIN {X 0,Y 345.777,Z 744.22,A -85,B 0,C 180,E1 801.018,E2 801.018} C_VEL
LIN {X 0,Y 343.344,Z 742.272,A -85,B 0,C 180,E1 798.75,E2 798.75} C_VEL
LIN {X 0,Y 338.087,Z 739.324,A -85,B 0,C 180,E1 795.792,E2 795.792} C_VEL
LIN {X 0,Y 331.784,Z 734.948,A -85,B 0,C 180,E1 792.463,E2 792.463} C_VEL
LIN {X 0,Y 328.202,Z 732.369,A -85,B 0,C 180,E1 790.793,E2 790.793} C_VEL
LIN {X 0,Y 318.811,Z 725.996,A -85,B 0,C 180,E1 787.117,E2 787.117} C_VEL
LIN {X 0,Y 313.742,Z 722.638,A -85,B 0,C 180,E1 785.271,E2 785.271} C_VEL
LIN {X 0,Y 302.178,Z 715.568,A -85,B 0,C 180,E1 781.268,E2 781.268} C_VEL
LIN {X 0,Y 289.124,Z 708.123,A -85,B 0,C 180,E1 776.816,E2 776.816} C_VEL
LIN {X 0,Y 277.681,Z 701.885,A -85,B 0,C 180,E1 772.73,E2 772.73} C_VEL
LIN {X 0,Y 264.103,Z 694.224,A -85,B 0,C 180,E1 767.264,E2 767.264} C_VEL
LIN {X 0,Y 246.325,Z 681.589,A -85,B 0,C 180,E1 757.509,E2 757.509} C_VEL
LIN {X 0,Y 239.079,Z 673.14,A -85,B 0,C 180,E1 750.992,E2 750.992} C_VEL
LIN {X 0,Y 223.806,Z 687.921,A -85,B 0,C 180,E1 752.406,E2 752.406} C_VEL
LIN {X 0,Y 205.817,Z 702.873,A -85,B 0,C 180,E1 754.333,E2 754.333} C_VEL
LIN {X 0,Y 188.996,Z 714.837,A -85,B 0,C 180,E1 756.481,E2 756.481} C_VEL
LIN {X 0,Y 172.449,Z 725.093,A -85,B 0,C 180,E1 759.027,E2 759.027} C_VEL
LIN {X 0,Y 152.754,Z 735.464,A -85,B 0,C 180,E1 762.86,E2 762.86} C_VEL
LIN {X 0,Y 135.578,Z 742.968,A -85,B 0,C 180,E1 767.281,E2 767.281} C_VEL
LIN {X 0,Y 120.982,Z 748.405,A -85,B 0,C 180,E1 772.301,E2 772.301} C_VEL
LIN {X 0,Y 104.766,Z 753.466,A -85,B 0,C 180,E1 780.286,E2 780.286} C_VEL
LIN {X 0,Y 90.938,Z 756.741,A -85,B 0,C 180,E1 791.409,E2 791.409} C_VEL
LIN {X 0,Y 82.781,Z 758.099,A -85,B 0,C 180,E1 803.76,E2 803.76} C_VEL
LIN {X 0,Y 80.721,Z 758.367,A -85,B 0,C 180,E1 810,E2 810} C_VEL
LIN {X 0,Y 87.592,Z 757.381,A -85,B 0,C 180,E1 824.543,E2 824.543} C_VEL
LIN {X 0,Y 98.607,Z 754.996,A -85,B 0,C 180,E1 835.515,E2 835.515} C_VEL
LIN {X 0,Y 112.616,Z 751.157,A -85,B 0,C 180,E1 844.006,E2 844.006} C_VEL
LIN {X 0,Y 131.427,Z 744.636,A -85,B 0,C 180,E1 851.437,E2 851.437} C_VEL
LIN {X 0,Y 147.519,Z 737.864,A -85,B 0,C 180,E1 855.921,E2 855.921} C_VEL
LIN {X 0,Y 165.629,Z 728.896,A -85,B 0,C 180,E1 859.763,E2 859.763} C_VEL
LIN {X 0,Y 185.287,Z 717.295,A -85,B 0,C 180,E1 862.993,E2 862.993} C_VEL
LIN {X 0,Y 202.057,Z 705.676,A -85,B 0,C 180,E1 865.22,E2 865.22} C_VEL
LIN {X 0,Y 218.102,Z 692.904,A -85,B 0,C 180,E1 867.019,E2 867.019} C_VEL
LIN {X 0,Y 236.202,Z 676.119,A -85,B 0,C 180,E1 868.759,E2 868.759} C_VEL
LIN {X 0,Y 239.127,Z 673.138,A -85,B 0,C 180,E1 868.989,E2 868.989} C_VEL
LIN {X 0,Y 251.29,Z 685.683,A -85,B 0,C 180,E1 859.265,E2 859.265} C_VEL
LIN {X 0,Y 269.997,Z 697.541,A -85,B 0,C 180,E1 850.28,E2 850.28} C_VEL
LIN {X 0,Y 284.137,Z 705.376,A -85,B 0,C 180,E1 844.921,E2 844.921} C_VEL
LIN {X 0,Y 293.581,Z 710.641,A -85,B 0,C 180,E1 841.629,E2 841.629} C_VEL
LIN {X 0,Y 305.12,Z 717.26,A -85,B 0,C 180,E1 837.728,E2 837.728} C_VEL
LIN {X 0,Y 316.707,Z 724.424,A -85,B 0,C 180,E1 833.712,E2 833.712} C_VEL
LIN {X 0,Y 325.937,Z 730.945,A -85,B 0,C 180,E1 830.093,E2 830.093} C_VEL
LIN {X 0,Y 330.579,Z 734.001,A -85,B 0,C 180,E1 828.149,E2 828.149} C_VEL
LIN {X 0,Y 337.041,Z 738.691,A -85,B 0,C 180,E1 824.779,E2 824.779} C_VEL
LIN {X 0,Y 342.884,Z 742.065,A -85,B 0,C 180,E1 821.531,E2 821.531} C_VEL
LIN {X 0,Y 344.992,Z 743.579,A -85,B 0,C 180,E1 819.794,E2 819.794} C_VEL
LIN {X 0,Y 347.725,Z 745.836,A -85,B 0,C 180,E1 816.604,E2 816.604} C_VEL
LIN {X 0,Y 349.474,Z 747.051,A -85,B 0,C 180,E1 813.773,E2 813.773} C_VEL
LIN {X 0,Y 349.976,Z 747.414,A -85,B 0,C 180,E1 812.57,E2 812.57} C_VEL
LIN {X 0,Y 349.497,Z 747.871,A -85,B 0,C 180,E1 811.397,E2 811.397} C_VEL
LIN {X 0,Y 346.597,Z 748.631,A -85,B 0,C 180,E1 809.72,E2 809.72} C_VEL
LIN {X 0,Y 342.453,Z 749.088,A -85,B 0,C 180,E1 807.46,E2 807.46} C_VEL
LIN {X 0,Y 341.921,Z 748.969,A -85,B 0,C 180,E1 806.803,E2 806.803} C_VEL
LIN {X 0,Y 340.409,Z 747.958,A -85,B 0,C 180,E1 804.1,E2 804.1} C_VEL
LIN {X 0,Y 337.871,Z 745.927,A -85,B 0,C 180,E1 800.977,E2 800.977} C_VEL
LIN {X 0,Y 335.43,Z 744.059,A -85,B 0,C 180,E1 798.829,E2 798.829} C_VEL
LIN {X 0,Y 329.617,Z 740.707,A -85,B 0,C 180,E1 795.599,E2 795.599} C_VEL
LIN {X 0,Y 323.285,Z 736.179,A -85,B 0,C 180,E1 792.292,E2 792.292} C_VEL
LIN {X 0,Y 318.577,Z 733.075,A -85,B 0,C 180,E1 790.32,E2 790.32} C_VEL
LIN {X 0,Y 308.704,Z 726.513,A -85,B 0,C 180,E1 786.439,E2 786.439} C_VEL
LIN {X 0,Y 296.372,Z 719.279,A -85,B 0,C 180,E1 782.12,E2 782.12} C_VEL
LIN {X 0,Y 282.592,Z 711.846,A -85,B 0,C 180,E1 777.364,E2 777.364} C_VEL
LIN {X 0,Y 271.061,Z 705.855,A -85,B 0,C 180,E1 773.175,E2 773.175} C_VEL
LIN {X 0,Y 257.916,Z 698.767,A -85,B 0,C 180,E1 767.772,E2 767.772} C_VEL
LIN {X 0,Y 238.866,Z 685.324,A -85,B 0,C 180,E1 756.77,E2 756.77} C_VEL
LIN {X 0,Y 234.953,Z 681.432,A -85,B 0,C 180,E1 753.433,E2 753.433} C_VEL
LIN {X 0,Y 220.752,Z 694.313,A -85,B 0,C 180,E1 754.943,E2 754.943} C_VEL
LIN {X 0,Y 204.028,Z 707.603,A -85,B 0,C 180,E1 756.993,E2 756.993} C_VEL
LIN {X 0,Y 184.869,Z 720.575,A -85,B 0,C 180,E1 759.833,E2 759.833} C_VEL
LIN {X 0,Y 168.841,Z 729.879,A -85,B 0,C 180,E1 762.757,E2 762.757} C_VEL
LIN {X 0,Y 151.625,Z 738.489,A -85,B 0,C 180,E1 766.707,E2 766.707} C_VEL
LIN {X 0,Y 132.926,Z 746.312,A -85,B 0,C 180,E1 772.468,E2 772.468} C_VEL
LIN {X 0,Y 117.377,Z 751.612,A -85,B 0,C 180,E1 779.267,E2 779.267} C_VEL
LIN {X 0,Y 104.016,Z 755.344,A -85,B 0,C 180,E1 787.985,E2 787.985} C_VEL
LIN {X 0,Y 92.786,Z 757.724,A -85,B 0,C 180,E1 800.699,E2 800.699} C_VEL
LIN {X 0,Y 88.827,Z 758.19,A -85,B 0,C 180,E1 810,E2 810} C_VEL
LIN {X 0,Y 95.612,Z 757.183,A -85,B 0,C 180,E1 823.449,E2 823.449} C_VEL
LIN {X 0,Y 106.35,Z 754.743,A -85,B 0,C 180,E1 833.843,E2 833.843} C_VEL
LIN {X 0,Y 120.196,Z 750.759,A -85,B 0,C 180,E1 842.163,E2 842.163} C_VEL
LIN {X 0,Y 138.464,Z 744.128,A -85,B 0,C 180,E1 849.449,E2 849.449} C_VEL
LIN {X 0,Y 154.16,Z 737.288,A -85,B 0,C 180,E1 853.941,E2 853.941} C_VEL
LIN {X 0,Y 171.48,Z 728.47,A -85,B 0,C 180,E1 857.768,E2 857.768} C_VEL
LIN {X 0,Y 191.21,Z 716.507,A -85,B 0,C 180,E1 861.174,E2 861.174} C_VEL
LIN {X 0,Y 206.802,Z 705.502,A -85,B 0,C 180,E1 863.37,E2 863.37} C_VEL
LIN {X 0,Y 222.625,Z 692.726,A -85,B 0,C 180,E1 865.266,E2 865.266} C_VEL
LIN {X 0,Y 235.143,Z 681.375,A -85,B 0,C 180,E1 866.523,E2 866.523} C_VEL
LIN {X 0,Y 249.838,Z 693.856,A -85,B 0,C 180,E1 856.182,E2 856.182} C_VEL
LIN {X 0,Y 266.874,Z 703.656,A -85,B 0,C 180,E1 848.459,E2 848.459} C_VEL
LIN {X 0,Y 278.132,Z 709.563,A -85,B 0,C 180,E1 844.223,E2 844.223} C_VEL
LIN {X 0,Y 287.658,Z 714.627,A -85,B 0,C 180,E1 840.844,E2 840.844} C_VEL
LIN {X 0,Y 298.685,Z 720.653,A -85,B 0,C 180,E1 837.067,E2 837.067} C_VEL
LIN {X 0,Y 309.883,Z 727.261,A -85,B 0,C 180,E1 833.132,E2 833.132} C_VEL
LIN {X 0,Y 320.375,Z 734.171,A -85,B 0,C 180,E1 828.974,E2 828.974} C_VEL
LIN {X 0,Y 323.845,Z 736.621,A -85,B 0,C 180,E1 827.425,E2 827.425} C_VEL
LIN {X 0,Y 330.33,Z 741.149,A -85,B 0,C 180,E1 824.012,E2 824.012} C_VEL
LIN {X 0,Y 335.736,Z 744.207,A -85,B 0,C 180,E1 820.987,E2 820.987} C_VEL
LIN {X 0,Y 338.505,Z 746.501,A -85,B 0,C 180,E1 818.294,E2 818.294} C_VEL
LIN {X 0,Y 340.742,Z 748.155,A -85,B 0,C 180,E1 815.387,E2 815.387} C_VEL
LIN {X 0,Y 342.174,Z 749.126,A -85,B 0,C 180,E1 812.497,E2 812.497} C_VEL
LIN {X 0,Y 342.582,Z 749.319,A -85,B 0,C 180,E1 809.666,E2 809.666} C_VEL
LIN {X 0,Y 342.061,Z 749.031,A -85,B 0,C 180,E1 807.152,E2 807.152} C_VEL
LIN {X 0,Y 341.921,Z 748.969,A -85,B 0,C 180,E1 806.803,E2 806.803} C_VEL
LIN {X 0,Y 340.476,Z 748.805,A -85,B 0,C 180,E1 805.62,E2 805.62} C_VEL
LIN {X 0,Y 336.128,Z 748.609,A -85,B 0,C 180,E1 803.875,E2 803.875} C_VEL
LIN {X 0,Y 331.044,Z 747.898,A -85,B 0,C 180,E1 801.821,E2 801.821} C_VEL
LIN {X 0,Y 329.997,Z 747.368,A -85,B 0,C 180,E1 801.065,E2 801.065} C_VEL
LIN {X 0,Y 327.743,Z 745.685,A -85,B 0,C 180,E1 799.098,E2 799.098} C_VEL
LIN {X 0,Y 322.131,Z 742.444,A -85,B 0,C 180,E1 795.991,E2 795.991} C_VEL
LIN {X 0,Y 315.507,Z 737.715,A -85,B 0,C 180,E1 792.538,E2 792.538} C_VEL
LIN {X 0,Y 307.962,Z 733.069,A -85,B 0,C 180,E1 789.476,E2 789.476} C_VEL
LIN {X 0,Y 300.906,Z 728.661,A -85,B 0,C 180,E1 786.711,E2 786.711} C_VEL
LIN {X 0,Y 288.799,Z 722.046,A -85,B 0,C 180,E1 782.416,E2 782.416} C_VEL
LIN {X 0,Y 275.553,Z 715.245,A -85,B 0,C 180,E1 777.769,E2 777.769} C_VEL
LIN {X 0,Y 264.138,Z 709.611,A -85,B 0,C 180,E1 773.542,E2 773.542} C_VEL
LIN {X 0,Y 248.446,Z 701.287,A -85,B 0,C 180,E1 766.757,E2 766.757} C_VEL
LIN {X 0,Y 231.378,Z 689.03,A -85,B 0,C 180,E1 755.957,E2 755.957} C_VEL
LIN {X 0,Y 214.487,Z 703.226,A -85,B 0,C 180,E1 758.026,E2 758.026} C_VEL
LIN {X 0,Y 198.208,Z 715.105,A -85,B 0,C 180,E1 760.391,E2 760.391} C_VEL
LIN {X 0,Y 180.535,Z 726.321,A -85,B 0,C 180,E1 763.494,E2 763.494} C_VEL
LIN {X 0,Y 162.63,Z 735.913,A -85,B 0,C 180,E1 767.451,E2 767.451} C_VEL
LIN {X 0,Y 147.217,Z 742.949,A -85,B 0,C 180,E1 771.831,E2 771.831} C_VEL
LIN {X 0,Y 132.845,Z 748.594,A -85,B 0,C 180,E1 777.19,E2 777.19} C_VEL
LIN {X 0,Y 117.427,Z 753.626,A -85,B 0,C 180,E1 785.343,E2 785.343} C_VEL
LIN {X 0,Y 105.346,Z 756.628,A -85,B 0,C 180,E1 795.497,E2 795.497} C_VEL
LIN {X 0,Y 98.438,Z 757.812,A -85,B 0,C 180,E1 805.923,E2 805.923} C_VEL
LIN {X 0,Y 96.99,Z 758.01,A -85,B 0,C 180,E1 810.166,E2 810.166} C_VEL
LIN {X 0,Y 103.878,Z 756.938,A -85,B 0,C 180,E1 822.789,E2 822.789} C_VEL
LIN {X 0,Y 114.453,Z 754.417,A -85,B 0,C 180,E1 832.603,E2 832.603} C_VEL
LIN {X 0,Y 128.58,Z 750.124,A -85,B 0,C 180,E1 840.875,E2 840.875} C_VEL
LIN {X 0,Y 144.869,Z 743.95,A -85,B 0,C 180,E1 847.394,E2 847.394} C_VEL
LIN {X 0,Y 160.141,Z 737.113,A -85,B 0,C 180,E1 851.913,E2 851.913} C_VEL
LIN {X 0,Y 177.065,Z 728.291,A -85,B 0,C 180,E1 855.813,E2 855.813} C_VEL
LIN {X 0,Y 196.417,Z 716.329,A -85,B 0,C 180,E1 859.324,E2 859.324} C_VEL
LIN {X 0,Y 211.752,Z 705.328,A -85,B 0,C 180,E1 861.605,E2 861.605} C_VEL
LIN {X 0,Y 227.47,Z 692.439,A -85,B 0,C 180,E1 863.6,E2 863.6} C_VEL
LIN {X 0,Y 231.416,Z 689.065,A -85,B 0,C 180,E1 864.011,E2 864.011} C_VEL
LIN {X 0,Y 250.266,Z 702.367,A -85,B 0,C 180,E1 852.342,E2 852.342} C_VEL
LIN {X 0,Y 264.427,Z 709.745,A -85,B 0,C 180,E1 846.348,E2 846.348} C_VEL
LIN {X 0,Y 276.687,Z 715.807,A -85,B 0,C 180,E1 841.839,E2 841.839} C_VEL
LIN {X 0,Y 291.272,Z 723.322,A -85,B 0,C 180,E1 836.721,E2 836.721} C_VEL
LIN {X 0,Y 302.474,Z 729.498,A -85,B 0,C 180,E1 832.736,E2 832.736} C_VEL
LIN {X 0,Y 312.113,Z 735.562,A -85,B 0,C 180,E1 828.876,E2 828.876} C_VEL
LIN {X 0,Y 316.064,Z 738.128,A -85,B 0,C 180,E1 827.176,E2 827.176} C_VEL
LIN {X 0,Y 322.373,Z 742.584,A -85,B 0,C 180,E1 823.875,E2 823.875} C_VEL
LIN {X 0,Y 328.05,Z 745.816,A -85,B 0,C 180,E1 820.714,E2 820.714} C_VEL
LIN {X 0,Y 330.674,Z 747.976,A -85,B 0,C 180,E1 818.169,E2 818.169} C_VEL
LIN {X 0,Y 332.976,Z 749.68,A -85,B 0,C 180,E1 815.168,E2 815.168} C_VEL
LIN {X 0,Y 334.397,Z 750.624,A -85,B 0,C 180,E1 812.227,E2 812.227} C_VEL
LIN {X 0,Y 334.717,Z 750.791,A -85,B 0,C 180,E1 809.658,E2 809.658} C_VEL
LIN {X 0,Y 334.152,Z 750.473,A -85,B 0,C 180,E1 807.085,E2 807.085} C_VEL
LIN {X 0,Y 332.619,Z 749.452,A -85,B 0,C 180,E1 804.283,E2 804.283} C_VEL
LIN {X 0,Y 329.997,Z 747.368,A -85,B 0,C 180,E1 801.065,E2 801.065} C_VEL
LIN {X 0,Y 327.997,Z 746.602,A -85,B 0,C 180,E1 799.974,E2 799.974} C_VEL
LIN {X 0,Y 323.165,Z 745.657,A -85,B 0,C 180,E1 798.547,E2 798.547} C_VEL
LIN {X 0,Y 314.967,Z 743.739,A -85,B 0,C 180,E1 796.357,E2 796.357} C_VEL
LIN {X 0,Y 312.927,Z 742.737,A -85,B 0,C 180,E1 795.52,E2 795.52} C_VEL
LIN {X 0,Y 307.121,Z 738.708,A -85,B 0,C 180,E1 792.538,E2 792.538} C_VEL
LIN {X 0,Y 296.245,Z 732.467,A -85,B 0,C 180,E1 788.154,E2 788.154} C_VEL
LIN {X 0,Y 284.667,Z 726.346,A -85,B 0,C 180,E1 783.96,E2 783.96} C_VEL
LIN {X 0,Y 271.22,Z 719.708,A -85,B 0,C 180,E1 779.178,E2 779.178} C_VEL
LIN {X 0,Y 258.276,Z 713.677,A -85,B 0,C 180,E1 774.39,E2 774.39} C_VEL
LIN {X 0,Y 244.901,Z 707.135,A -85,B 0,C 180,E1 768.698,E2 768.698} C_VEL
LIN {X 0,Y 227.707,Z 696.337,A -85,B 0,C 180,E1 758.601,E2 758.601} C_VEL
LIN {X 0,Y 210.641,Z 709.936,A -85,B 0,C 180,E1 761.005,E2 761.005} C_VEL
LIN {X 0,Y 193.971,Z 721.318,A -85,B 0,C 180,E1 763.815,E2 763.815} C_VEL
LIN {X 0,Y 177.802,Z 730.934,A -85,B 0,C 180,E1 767.128,E2 767.128} C_VEL
LIN {X 0,Y 160.722,Z 739.673,A -85,B 0,C 180,E1 771.535,E2 771.535} C_VEL
LIN {X 0,Y 144.054,Z 746.788,A -85,B 0,C 180,E1 777.226,E2 777.226} C_VEL
LIN {X 0,Y 130.422,Z 751.68,A -85,B 0,C 180,E1 783.602,E2 783.602} C_VEL
LIN {X 0,Y 117.783,Z 755.419,A -85,B 0,C 180,E1 792.208,E2 792.208} C_VEL
LIN {X 0,Y 107.949,Z 757.47,A -85,B 0,C 180,E1 803.619,E2 803.619} C_VEL
LIN {X 0,Y 105.06,Z 757.836,A -85,B 0,C 180,E1 810,E2 810} C_VEL
LIN {X 0,Y 111.852,Z 756.763,A -85,B 0,C 180,E1 821.863,E2 821.863} C_VEL
LIN {X 0,Y 122.041,Z 754.241,A -85,B 0,C 180,E1 831.128,E2 831.128} C_VEL
LIN {X 0,Y 135.666,Z 749.944,A -85,B 0,C 180,E1 839.102,E2 839.102} C_VEL
LIN {X 0,Y 151.446,Z 743.771,A -85,B 0,C 180,E1 845.516,E2 845.516} C_VEL
LIN {X 0,Y 166.308,Z 736.938,A -85,B 0,C 180,E1 850.033,E2 850.033} C_VEL
LIN {X 0,Y 182.844,Z 728.111,A -85,B 0,C 180,E1 853.98,E2 853.98} C_VEL
LIN {X 0,Y 201.817,Z 716.152,A -85,B 0,C 180,E1 857.571,E2 857.571} C_VEL
LIN {X 0,Y 217.79,Z 704.454,A -85,B 0,C 180,E1 860.05,E2 860.05} C_VEL
LIN {X 0,Y 227.762,Z 696.335,A -85,B 0,C 180,E1 861.382,E2 861.382} C_VEL
LIN {X 0,Y 246.356,Z 707.894,A -85,B 0,C 180,E1 850.625,E2 850.625} C_VEL
LIN {X 0,Y 261.635,Z 715.19,A -85,B 0,C 180,E1 844.362,E2 844.362} C_VEL
LIN {X 0,Y 273.524,Z 720.912,A -85,B 0,C 180,E1 839.96,E2 839.96} C_VEL
LIN {X 0,Y 284.787,Z 726.411,A -85,B 0,C 180,E1 835.996,E2 835.996} C_VEL
LIN {X 0,Y 296.245,Z 732.466,A -85,B 0,C 180,E1 831.846,E2 831.846} C_VEL
LIN {X 0,Y 307.122,Z 738.707,A -85,B 0,C 180,E1 827.462,E2 827.462} C_VEL
LIN {X 0,Y 313.029,Z 742.806,A -85,B 0,C 180,E1 824.425,E2 824.425} C_VEL
LIN {X 0,Y 319.021,Z 746.466,A -85,B 0,C 180,E1 821.18,E2 821.18} C_VEL
LIN {X 0,Y 321.038,Z 747.652,A -85,B 0,C 180,E1 819.862,E2 819.862} C_VEL
LIN {X 0,Y 323.709,Z 749.886,A -85,B 0,C 180,E1 816.918,E2 816.918} C_VEL
LIN {X 0,Y 325.771,Z 751.282,A -85,B 0,C 180,E1 813.871,E2 813.871} C_VEL
LIN {X 0,Y 326.675,Z 751.853,A -85,B 0,C 180,E1 811.228,E2 811.228} C_VEL
LIN {X 0,Y 326.733,Z 751.873,A -85,B 0,C 180,E1 808.948,E2 808.948} C_VEL
LIN {X 0,Y 325.877,Z 751.363,A -85,B 0,C 180,E1 806.306,E2 806.306} C_VEL
LIN {X 0,Y 324.004,Z 750.115,A -85,B 0,C 180,E1 803.444,E2 803.444} C_VEL
LIN {X 0,Y 321.39,Z 747.946,A -85,B 0,C 180,E1 800.483,E2 800.483} C_VEL
LIN {X 0,Y 319.651,Z 746.811,A -85,B 0,C 180,E1 799.178,E2 799.178} C_VEL
LIN {X 0,Y 313.815,Z 743.32,A -85,B 0,C 180,E1 795.988,E2 795.988} C_VEL
LIN {X 0,Y 312.927,Z 742.737,A -85,B 0,C 180,E1 795.52,E2 795.52} C_VEL
LIN {X 0,Y 309.733,Z 741.395,A -85,B 0,C 180,E1 794.358,E2 794.358} C_VEL
LIN {X 0,Y 303.174,Z 739.768,A -85,B 0,C 180,E1 792.822,E2 792.822} C_VEL
LIN {X 0,Y 294.318,Z 737.42,A -85,B 0,C 180,E1 790.742,E2 790.742} C_VEL
LIN {X 0,Y 292.418,Z 736.53,A -85,B 0,C 180,E1 790.086,E2 790.086} C_VEL
LIN {X 0,Y 286.387,Z 733.313,A -85,B 0,C 180,E1 787.702,E2 787.702} C_VEL
LIN {X 0,Y 275.365,Z 727.97,A -85,B 0,C 180,E1 783.709,E2 783.709} C_VEL
LIN {X 0,Y 262.356,Z 722.047,A -85,B 0,C 180,E1 779.04,E2 779.04} C_VEL
LIN {X 0,Y 251.001,Z 717.048,A -85,B 0,C 180,E1 774.722,E2 774.722} C_VEL
LIN {X 0,Y 234.683,Z 709.175,A -85,B 0,C 180,E1 767.364,E2 767.364} C_VEL
LIN {X 0,Y 224.362,Z 703.273,A -85,B 0,C 180,E1 761.362,E2 761.362} C_VEL
LIN {X 0,Y 209.122,Z 714.754,A -85,B 0,C 180,E1 763.79,E2 763.79} C_VEL
LIN {X 0,Y 192.123,Z 725.961,A -85,B 0,C 180,E1 767.024,E2 767.024} C_VEL
LIN {X 0,Y 175.009,Z 735.562,A -85,B 0,C 180,E1 771.069,E2 771.069} C_VEL
LIN {X 0,Y 160.035,Z 742.754,A -85,B 0,C 180,E1 775.561,E2 775.561} C_VEL
LIN {X 0,Y 145.512,Z 748.783,A -85,B 0,C 180,E1 781.253,E2 781.253} C_VEL
LIN {X 0,Y 130.79,Z 753.765,A -85,B 0,C 180,E1 789.414,E2 789.414} C_VEL
LIN {X 0,Y 120.248,Z 756.495,A -85,B 0,C 180,E1 798.49,E2 798.49} C_VEL
LIN {X 0,Y 113.76,Z 757.58,A -85,B 0,C 180,E1 808.489,E2 808.489} C_VEL
LIN {X 0,Y 113.181,Z 757.658,A -85,B 0,C 180,E1 810,E2 810} C_VEL
LIN {X 0,Y 119.853,Z 756.587,A -85,B 0,C 180,E1 821.061,E2 821.061} C_VEL
LIN {X 0,Y 129.702,Z 754.065,A -85,B 0,C 180,E1 829.825,E2 829.825} C_VEL
LIN {X 0,Y 142.87,Z 749.763,A -85,B 0,C 180,E1 837.506,E2 837.506} C_VEL
LIN {X 0,Y 158.171,Z 743.593,A -85,B 0,C 180,E1 843.795,E2 843.795} C_VEL
LIN {X 0,Y 172.64,Z 736.762,A -85,B 0,C 180,E1 848.289,E2 848.289} C_VEL
LIN {X 0,Y 188.797,Z 727.931,A -85,B 0,C 180,E1 852.261,E2 852.261} C_VEL
LIN {X 0,Y 207.396,Z 715.974,A -85,B 0,C 180,E1 855.911,E2 855.911} C_VEL
LIN {X 0,Y 223.148,Z 704.236,A -85,B 0,C 180,E1 858.458,E2 858.458} C_VEL
LIN {X 0,Y 224.554,Z 703.226,A -85,B 0,C 180,E1 858.606,E2 858.606} C_VEL
LIN {X 0,Y 241.546,Z 712.644,A -85,B 0,C 180,E1 849.277,E2 849.277} C_VEL
LIN {X 0,Y 257.184,Z 719.714,A -85,B 0,C 180,E1 842.883,E2 842.883} C_VEL
LIN {X 0,Y 267.489,Z 724.392,A -85,B 0,C 180,E1 839.07,E2 839.07} C_VEL
LIN {X 0,Y 278.435,Z 729.417,A -85,B 0,C 180,E1 835.182,E2 835.182} C_VEL
LIN {X 0,Y 289.078,Z 734.623,A -85,B 0,C 180,E1 831.293,E2 831.293} C_VEL
LIN {X 0,Y 298.846,Z 739.909,A -85,B 0,C 180,E1 827.322,E2 827.322} C_VEL
LIN {X 0,Y 303.421,Z 742.763,A -85,B 0,C 180,E1 825.082,E2 825.082} C_VEL
LIN {X 0,Y 309.525,Z 746.46,A -85,B 0,C 180,E1 821.814,E2 821.814} C_VEL
LIN {X 0,Y 313.074,Z 748.438,A -85,B 0,C 180,E1 819.744,E2 819.744} C_VEL
LIN {X 0,Y 315.678,Z 750.643,A -85,B 0,C 180,E1 816.912,E2 816.912} C_VEL
LIN {X 0,Y 317.734,Z 752.042,A -85,B 0,C 180,E1 813.969,E2 813.969} C_VEL
LIN {X 0,Y 318.709,Z 752.655,A -85,B 0,C 180,E1 811.258,E2 811.258} C_VEL
LIN {X 0,Y 318.768,Z 752.679,A -85,B 0,C 180,E1 808.922,E2 808.922} C_VEL
LIN {X 0,Y 317.848,Z 752.12,A -85,B 0,C 180,E1 806.213,E2 806.213} C_VEL
LIN {X 0,Y 315.835,Z 750.759,A -85,B 0,C 180,E1 803.274,E2 803.274} C_VEL
LIN {X 0,Y 313.271,Z 748.61,A -85,B 0,C 180,E1 800.448,E2 800.448} C_VEL
LIN {X 0,Y 310.041,Z 746.75,A -85,B 0,C 180,E1 798.468,E2 798.468} C_VEL
LIN {X 0,Y 304.014,Z 743.137,A -85,B 0,C 180,E1 795.23,E2 795.23} C_VEL
LIN {X 0,Y 299.277,Z 740.131,A -85,B 0,C 180,E1 792.85,E2 792.85} C_VEL
LIN {X 0,Y 292.418,Z 736.53,A -85,B 0,C 180,E1 790.086,E2 790.086} C_VEL
LIN {X 0,Y 288.587,Z 735.08,A -85,B 0,C 180,E1 788.921,E2 788.921} C_VEL
LIN {X 0,Y 280.916,Z 733.569,A -85,B 0,C 180,E1 787.317,E2 787.317} C_VEL
LIN {X 0,Y 271.543,Z 731.725,A -85,B 0,C 180,E1 785.314,E2 785.314} C_VEL
LIN {X 0,Y 269.304,Z 730.966,A -85,B 0,C 180,E1 784.644,E2 784.644} C_VEL
LIN {X 0,Y 255.613,Z 725.169,A -85,B 0,C 180,E1 779.699,E2 779.699} C_VEL
LIN {X 0,Y 244.189,Z 720.411,A -85,B 0,C 180,E1 775.313,E2 775.313} C_VEL
LIN {X 0,Y 231.211,Z 714.676,A -85,B 0,C 180,E1 769.564,E2 769.564} C_VEL
LIN {X 0,Y 221.542,Z 709.675,A -85,B 0,C 180,E1 764.204,E2 764.204} C_VEL
LIN {X 0,Y 205.585,Z 720.963,A -85,B 0,C 180,E1 767.093,E2 767.093} C_VEL
LIN {X 0,Y 190.082,Z 730.585,A -85,B 0,C 180,E1 770.475,E2 770.475} C_VEL
LIN {X 0,Y 173.811,Z 739.313,A -85,B 0,C 180,E1 774.887,E2 774.887} C_VEL
LIN {X 0,Y 158.053,Z 746.43,A -85,B 0,C 180,E1 780.437,E2 780.437} C_VEL
LIN {X 0,Y 145.258,Z 751.328,A -85,B 0,C 180,E1 786.472,E2 786.472} C_VEL
LIN {X 0,Y 133.444,Z 755.057,A -85,B 0,C 180,E1 794.353,E2 794.353} C_VEL
LIN {X 0,Y 124.161,Z 757.117,A -85,B 0,C 180,E1 804.455,E2 804.455} C_VEL
LIN {X 0,Y 121.305,Z 757.48,A -85,B 0,C 180,E1 810,E2 810} C_VEL
LIN {X 0,Y 127.875,Z 756.411,A -85,B 0,C 180,E1 820.359,E2 820.359} C_VEL
LIN {X 0,Y 137.947,Z 753.739,A -85,B 0,C 180,E1 829.034,E2 829.034} C_VEL
LIN {X 0,Y 152.087,Z 748.878,A -85,B 0,C 180,E1 836.973,E2 836.973} C_VEL
LIN {X 0,Y 166.461,Z 742.753,A -85,B 0,C 180,E1 842.72,E2 842.72} C_VEL
LIN {X 0,Y 181.432,Z 735.387,A -85,B 0,C 180,E1 847.311,E2 847.311} C_VEL
LIN {X 0,Y 199.225,Z 725.133,A -85,B 0,C 180,E1 851.598,E2 851.598} C_VEL
LIN {X 0,Y 215.679,Z 713.96,A -85,B 0,C 180,E1 854.795,E2 854.795} C_VEL
LIN {X 0,Y 221.549,Z 709.68,A -85,B 0,C 180,E1 855.79,E2 855.79} C_VEL
LIN {X 0,Y 239.955,Z 718.593,A -85,B 0,C 180,E1 846.464,E2 846.464} C_VEL
LIN {X 0,Y 252.296,Z 723.83,A -85,B 0,C 180,E1 841.538,E2 841.538} C_VEL
LIN {X 0,Y 261.702,Z 727.815,A -85,B 0,C 180,E1 838.044,E2 838.044} C_VEL
LIN {X 0,Y 271.505,Z 731.988,A -85,B 0,C 180,E1 834.544,E2 834.544} C_VEL
LIN {X 0,Y 282.086,Z 736.827,A -85,B 0,C 180,E1 830.645,E2 830.645} C_VEL
LIN {X 0,Y 292.778,Z 742.195,A -85,B 0,C 180,E1 826.261,E2 826.261} C_VEL
LIN {X 0,Y 299.842,Z 746.328,A -85,B 0,C 180,E1 822.517,E2 822.517} C_VEL
LIN {X 0,Y 305.176,Z 749.07,A -85,B 0,C 180,E1 819.526,E2 819.526} C_VEL
LIN {X 0,Y 307.61,Z 751.026,A -85,B 0,C 180,E1 816.907,E2 816.907} C_VEL
LIN {X 0,Y 309.654,Z 752.449,A -85,B 0,C 180,E1 814.073,E2 814.073} C_VEL
LIN {X 0,Y 310.689,Z 753.105,A -85,B 0,C 180,E1 811.475,E2 811.475} C_VEL
LIN {X 0,Y 310.816,Z 753.204,A -85,B 0,C 180,E1 809.263,E2 809.263} C_VEL
LIN {X 0,Y 310.049,Z 752.723,A -85,B 0,C 180,E1 806.673,E2 806.673} C_VEL
LIN {X 0,Y 308.23,Z 751.493,A -85,B 0,C 180,E1 803.856,E2 803.856} C_VEL
LIN {X 0,Y 305.726,Z 749.515,A -85,B 0,C 180,E1 801.007,E2 801.007} C_VEL
LIN {X 0,Y 303.649,Z 748.348,A -85,B 0,C 180,E1 799.567,E2 799.567} C_VEL
LIN {X 0,Y 296.625,Z 744.515,A -85,B 0,C 180,E1 795.757,E2 795.757} C_VEL
LIN {X 0,Y 291.651,Z 741.665,A -85,B 0,C 180,E1 793.265,E2 793.265} C_VEL
LIN {X 0,Y 280.862,Z 736.188,A -85,B 0,C 180,E1 788.866,E2 788.866} C_VEL
LIN {X 0,Y 269.304,Z 730.966,A -85,B 0,C 180,E1 784.644,E2 784.644} C_VEL
LIN {X 0,Y 264.507,Z 729.706,A -85,B 0,C 180,E1 783.36,E2 783.36} C_VEL
LIN {X 0,Y 247.802,Z 727.506,A -85,B 0,C 180,E1 779.848,E2 779.848} C_VEL
LIN {X 0,Y 244.912,Z 726.631,A -85,B 0,C 180,E1 778.911,E2 778.911} C_VEL
LIN {X 0,Y 229.952,Z 720.634,A -85,B 0,C 180,E1 772.725,E2 772.725} C_VEL
LIN {X 0,Y 218.818,Z 715.775,A -85,B 0,C 180,E1 767.189,E2 767.189} C_VEL
LIN {X 0,Y 200.97,Z 727.693,A -85,B 0,C 180,E1 770.91,E2 770.91} C_VEL
LIN {X 0,Y 184.985,Z 736.811,A -85,B 0,C 180,E1 775.049,E2 775.049} C_VEL
LIN {X 0,Y 169.924,Z 744.225,A -85,B 0,C 180,E1 779.994,E2 779.994} C_VEL
LIN {X 0,Y 155.141,Z 750.311,A -85,B 0,C 180,E1 786.451,E2 786.451} C_VEL
LIN {X 0,Y 143.217,Z 754.316,A -85,B 0,C 180,E1 793.786,E2 793.786} C_VEL
LIN {X 0,Y 133.819,Z 756.716,A -85,B 0,C 180,E1 802.703,E2 802.703} C_VEL
LIN {X 0,Y 129.434,Z 757.303,A -85,B 0,C 180,E1 810,E2 810} C_VEL
LIN {X 0,Y 135.966,Z 756.223,A -85,B 0,C 180,E1 819.792,E2 819.792} C_VEL
LIN {X 0,Y 145.703,Z 753.564,A -85,B 0,C 180,E1 827.985,E2 827.985} C_VEL
LIN {X 0,Y 159.419,Z 748.701,A -85,B 0,C 180,E1 835.64,E2 835.64} C_VEL
LIN {X 0,Y 173.394,Z 742.576,A -85,B 0,C 180,E1 841.26,E2 841.26} C_VEL
LIN {X 0,Y 187.989,Z 735.211,A -85,B 0,C 180,E1 845.803,E2 845.803} C_VEL
LIN {X 0,Y 205.15,Z 725.108,A -85,B 0,C 180,E1 850.036,E2 850.036} C_VEL
LIN {X 0,Y 219.001,Z 715.741,A -85,B 0,C 180,E1 852.785,E2 852.785} C_VEL
LIN {X 0,Y 235.882,Z 723.122,A -85,B 0,C 180,E1 844.679,E2 844.679} C_VEL
LIN {X 0,Y 246.821,Z 727.399,A -85,B 0,C 180,E1 840.358,E2 840.358} C_VEL
LIN {X 0,Y 255.981,Z 731.023,A -85,B 0,C 180,E1 836.939,E2 836.939} C_VEL
LIN {X 0,Y 265.206,Z 734.706,A -85,B 0,C 180,E1 833.627,E2 833.627} C_VEL
LIN {X 0,Y 275.056,Z 738.868,A -85,B 0,C 180,E1 829.978,E2 829.978} C_VEL
LIN {X 0,Y 285.029,Z 743.44,A -85,B 0,C 180,E1 825.878,E2 825.878} C_VEL
LIN {X 0,Y 291.089,Z 746.743,A -85,B 0,C 180,E1 822.698,E2 822.698} C_VEL
LIN {X 0,Y 296.99,Z 749.557,A -85,B 0,C 180,E1 819.439,E2 819.439} C_VEL
LIN {X 0,Y 299.37,Z 751.21,A -85,B 0,C 180,E1 817.098,E2 817.098} C_VEL
LIN {X 0,Y 301.545,Z 752.65,A -85,B 0,C 180,E1 814.183,E2 814.183} C_VEL
LIN {X 0,Y 302.681,Z 753.331,A -85,B 0,C 180,E1 811.514,E2 811.514} C_VEL
LIN {X 0,Y 302.816,Z 753.423,A -85,B 0,C 180,E1 809.243,E2 809.243} C_VEL
LIN {X 0,Y 301.982,Z 752.929,A -85,B 0,C 180,E1 806.584,E2 806.584} C_VEL
LIN {X 0,Y 300.017,Z 751.676,A -85,B 0,C 180,E1 803.687,E2 803.687} C_VEL
LIN {X 0,Y 297.402,Z 749.753,A -85,B 0,C 180,E1 800.812,E2 800.812} C_VEL
LIN {X 0,Y 291.726,Z 747.068,A -85,B 0,C 180,E1 797.645,E2 797.645} C_VEL
LIN {X 0,Y 285.545,Z 743.694,A -85,B 0,C 180,E1 794.359,E2 794.359} C_VEL
LIN {X 0,Y 276.32,Z 739.474,A -85,B 0,C 180,E1 790.557,E2 790.557} C_VEL
LIN {X 0,Y 271.23,Z 737.261,A -85,B 0,C 180,E1 788.598,E2 788.598} C_VEL
LIN {X 0,Y 261.466,Z 733.192,A -85,B 0,C 180,E1 785.003,E2 785.003} C_VEL
LIN {X 0,Y 248.816,Z 728.162,A -85,B 0,C 180,E1 780.382,E2 780.382} C_VEL
LIN {X 0,Y 244.912,Z 726.631,A -85,B 0,C 180,E1 778.911,E2 778.911} C_VEL
LIN {X 0,Y 240.236,Z 725.485,A -85,B 0,C 180,E1 777.476,E2 777.476} C_VEL
LIN {X 0,Y 223.879,Z 723.986,A -85,B 0,C 180,E1 773.502,E2 773.502} C_VEL
LIN {X 0,Y 221.097,Z 723.221,A -85,B 0,C 180,E1 772.441,E2 772.441} C_VEL
LIN {X 0,Y 216.529,Z 721.476,A -85,B 0,C 180,E1 770.277,E2 770.277} C_VEL
LIN {X 0,Y 200.647,Z 731.616,A -85,B 0,C 180,E1 773.988,E2 773.988} C_VEL
LIN {X 0,Y 184.582,Z 740.393,A -85,B 0,C 180,E1 778.67,E2 778.67} C_VEL
LIN {X 0,Y 171.187,Z 746.624,A -85,B 0,C 180,E1 783.65,E2 783.65} C_VEL
LIN {X 0,Y 158.182,Z 751.817,A -85,B 0,C 180,E1 790.044,E2 790.044} C_VEL
LIN {X 0,Y 146.685,Z 755.418,A -85,B 0,C 180,E1 798.202,E2 798.202} C_VEL
LIN {X 0,Y 139.585,Z 756.864,A -85,B 0,C 180,E1 806.304,E2 806.304} C_VEL
LIN {X 0,Y 137.568,Z 757.125,A -85,B 0,C 180,E1 810,E2 810} C_VEL
LIN {X 0,Y 143.977,Z 756.059,A -85,B 0,C 180,E1 819.19,E2 819.19} C_VEL
LIN {X 0,Y 154.003,Z 753.237,A -85,B 0,C 180,E1 827.375,E2 827.375} C_VEL
LIN {X 0,Y 167.44,Z 748.253,A -85,B 0,C 180,E1 834.706,E2 834.706} C_VEL
LIN {X 0,Y 180.428,Z 742.398,A -85,B 0,C 180,E1 839.913,E2 839.913} C_VEL
LIN {X 0,Y 194.667,Z 735.036,A -85,B 0,C 180,E1 844.397,E2 844.397} C_VEL
LIN {X 0,Y 211.453,Z 724.929,A -85,B 0,C 180,E1 848.616,E2 848.616} C_VEL
LIN {X 0,Y 216.753,Z 721.398,A -85,B 0,C 180,E1 849.721,E2 849.721} C_VEL
LIN {X 0,Y 230.808,Z 726.929,A -85,B 0,C 180,E1 843.269,E2 843.269} C_VEL
LIN {X 0,Y 242.668,Z 731.213,A -85,B 0,C 180,E1 838.64,E2 838.64} C_VEL
LIN {X 0,Y 256.441,Z 736.237,A -85,B 0,C 180,E1 833.61,E2 833.61} C_VEL
LIN {X 0,Y 268.011,Z 740.766,A -85,B 0,C 180,E1 829.284,E2 829.284} C_VEL
LIN {X 0,Y 277.84,Z 744.94,A -85,B 0,C 180,E1 825.229,E2 825.229} C_VEL
LIN {X 0,Y 284.773,Z 748.398,A -85,B 0,C 180,E1 821.543,E2 821.543} C_VEL
LIN {X 0,Y 289.738,Z 750.516,A -85,B 0,C 180,E1 818.733,E2 818.733} C_VEL
LIN {X 0,Y 292.579,Z 752.412,A -85,B 0,C 180,E1 815.49,E2 815.49} C_VEL
LIN {X 0,Y 294.277,Z 753.384,A -85,B 0,C 180,E1 812.624,E2 812.624} C_VEL
LIN {X 0,Y 294.869,Z 753.67,A -85,B 0,C 180,E1 809.806,E2 809.806} C_VEL
LIN {X 0,Y 294.18,Z 753.317,A -85,B 0,C 180,E1 807.078,E2 807.078} C_VEL
LIN {X 0,Y 292.27,Z 752.209,A -85,B 0,C 180,E1 804.11,E2 804.11} C_VEL
LIN {X 0,Y 289.675,Z 750.467,A -85,B 0,C 180,E1 801.206,E2 801.206} C_VEL
LIN {X 0,Y 283.44,Z 747.736,A -85,B 0,C 180,E1 797.735,E2 797.735} C_VEL
LIN {X 0,Y 277.767,Z 744.906,A -85,B 0,C 180,E1 794.739,E2 794.739} C_VEL
LIN {X 0,Y 267.387,Z 740.476,A -85,B 0,C 180,E1 790.451,E2 790.451} C_VEL
LIN {X 0,Y 255.798,Z 736.003,A -85,B 0,C 180,E1 786.161,E2 786.161} C_VEL
LIN {X 0,Y 242.054,Z 730.999,A -85,B 0,C 180,E1 781.133,E2 781.133} C_VEL
LIN {X 0,Y 230.805,Z 726.931,A -85,B 0,C 180,E1 776.732,E2 776.732} C_VEL
LIN {X 0,Y 221.097,Z 723.221,A -85,B 0,C 180,E1 772.441,E2 772.441} C_VEL
LIN {X 0,Y 219.478,Z 723.419,A -85,B 0,C 180,E1 772.207,E2 772.207} C_VEL
LIN {X 0,Y 216.64,Z 724.602,A -85,B 0,C 180,E1 772.346,E2 772.346} C_VEL
LIN {X 0,Y 213.101,Z 726.692,A -85,B 0,C 180,E1 773.041,E2 773.041} C_VEL
LIN {X 0,Y 204.827,Z 732.894,A -85,B 0,C 180,E1 775.967,E2 775.967} C_VEL
LIN {X 0,Y 204.191,Z 733.282,A -85,B 0,C 180,E1 776.148,E2 776.148} C_VEL
LIN {X 0,Y 188.872,Z 741.565,A -85,B 0,C 180,E1 780.869,E2 780.869} C_VEL
LIN {X 0,Y 176.105,Z 747.533,A -85,B 0,C 180,E1 785.874,E2 785.874} C_VEL
LIN {X 0,Y 163.316,Z 752.541,A -85,B 0,C 180,E1 792.545,E2 792.545} C_VEL
LIN {X 0,Y 153.255,Z 755.581,A -85,B 0,C 180,E1 800.123,E2 800.123} C_VEL
LIN {X 0,Y 146.98,Z 756.783,A -85,B 0,C 180,E1 807.661,E2 807.661} C_VEL
LIN {X 0,Y 145.706,Z 756.947,A -85,B 0,C 180,E1 810,E2 810} C_VEL
LIN {X 0,Y 152.048,Z 755.883,A -85,B 0,C 180,E1 818.698,E2 818.698} C_VEL
LIN {X 0,Y 161.827,Z 753.062,A -85,B 0,C 180,E1 826.51,E2 826.51} C_VEL
LIN {X 0,Y 174.903,Z 748.076,A -85,B 0,C 180,E1 833.586,E2 833.586} C_VEL
LIN {X 0,Y 188.224,Z 741.888,A -85,B 0,C 180,E1 838.904,E2 838.904} C_VEL
LIN {X 0,Y 202.9,Z 734.055,A -85,B 0,C 180,E1 843.495,E2 843.495} C_VEL
LIN {X 0,Y 214.966,Z 726.715,A -85,B 0,C 180,E1 846.534,E2 846.534} C_VEL
LIN {X 0,Y 231.22,Z 732.337,A -85,B 0,C 180,E1 839.633,E2 839.633} C_VEL
LIN {X 0,Y 241.345,Z 735.769,A -85,B 0,C 180,E1 835.782,E2 835.782} C_VEL
LIN {X 0,Y 251.463,Z 739.205,A -85,B 0,C 180,E1 832.108,E2 832.108} C_VEL
LIN {X 0,Y 261.343,Z 742.773,A -85,B 0,C 180,E1 828.406,E2 828.406} C_VEL
LIN {X 0,Y 271.149,Z 746.543,A -85,B 0,C 180,E1 824.302,E2 824.302} C_VEL
LIN {X 0,Y 278.075,Z 749.597,A -85,B 0,C 180,E1 820.565,E2 820.565} C_VEL
LIN {X 0,Y 282.184,Z 751.233,A -85,B 0,C 180,E1 818.147,E2 818.147} C_VEL
LIN {X 0,Y 284.987,Z 752.872,A -85,B 0,C 180,E1 814.83,E2 814.83} C_VEL
LIN {X 0,Y 286.427,Z 753.615,A -85,B 0,C 180,E1 812.2,E2 812.2} C_VEL
LIN {X 0,Y 286.849,Z 753.821,A -85,B 0,C 180,E1 809.601,E2 809.601} C_VEL
LIN {X 0,Y 286.116,Z 753.495,A -85,B 0,C 180,E1 806.996,E2 806.996} C_VEL
LIN {X 0,Y 284.042,Z 752.392,A -85,B 0,C 180,E1 803.939,E2 803.939} C_VEL
LIN {X 0,Y 281.654,Z 750.995,A -85,B 0,C 180,E1 801.426,E2 801.426} C_VEL
LIN {X 0,Y 274.493,Z 748.098,A -85,B 0,C 180,E1 797.486,E2 797.486} C_VEL
LIN {X 0,Y 269.971,Z 746.105,A -85,B 0,C 180,E1 795.165,E2 795.165} C_VEL
LIN {X 0,Y 259.379,Z 742.006,A -85,B 0,C 180,E1 790.815,E2 790.815} C_VEL
LIN {X 0,Y 248.225,Z 738.095,A -85,B 0,C 180,E1 786.697,E2 786.697} C_VEL
LIN {X 0,Y 235.52,Z 733.802,A -85,B 0,C 180,E1 782.013,E2 782.013} C_VEL
LIN {X 0,Y 224.057,Z 729.956,A -85,B 0,C 180,E1 777.506,E2 777.506} C_VEL
LIN {X 0,Y 214.818,Z 726.719,A -85,B 0,C 180,E1 773.437,E2 773.437} C_VEL
LIN {X 0,Y 204.191,Z 733.282,A -85,B 0,C 180,E1 776.148,E2 776.148} C_VEL
LIN {X 0,Y 199.876,Z 736.259,A -85,B 0,C 180,E1 777.775,E2 777.775} C_VEL
LIN {X 0,Y 192.147,Z 743.06,A -85,B 0,C 180,E1 783.023,E2 783.023} C_VEL
LIN {X 0,Y 188.599,Z 745.079,A -85,B 0,C 180,E1 784.811,E2 784.811} C_VEL
LIN {X 0,Y 176.817,Z 750.204,A -85,B 0,C 180,E1 790.169,E2 790.169} C_VEL
LIN {X 0,Y 165.601,Z 754.207,A -85,B 0,C 180,E1 797.093,E2 797.093} C_VEL
LIN {X 0,Y 156.95,Z 756.377,A -85,B 0,C 180,E1 805.25,E2 805.25} C_VEL
LIN {X 0,Y 153.846,Z 756.769,A -85,B 0,C 180,E1 810,E2 810} C_VEL
LIN {X 0,Y 160.131,Z 755.707,A -85,B 0,C 180,E1 818.256,E2 818.256} C_VEL
LIN {X 0,Y 169.685,Z 752.886,A -85,B 0,C 180,E1 825.725,E2 825.725} C_VEL
LIN {X 0,Y 182.427,Z 747.9,A -85,B 0,C 180,E1 832.558,E2 832.558} C_VEL
LIN {X 0,Y 195.523,Z 741.656,A -85,B 0,C 180,E1 837.784,E2 837.784} C_VEL
LIN {X 0,Y 209.751,Z 733.875,A -85,B 0,C 180,E1 842.265,E2 842.265} C_VEL
LIN {X 0,Y 213.654,Z 731.623,A -85,B 0,C 180,E1 843.241,E2 843.241} C_VEL
LIN {X 0,Y 226.477,Z 735.642,A -85,B 0,C 180,E1 837.994,E2 837.994} C_VEL
LIN {X 0,Y 236.037,Z 738.656,A -85,B 0,C 180,E1 834.387,E2 834.387} C_VEL
LIN {X 0,Y 245.293,Z 741.466,A -85,B 0,C 180,E1 831.016,E2 831.016} C_VEL
LIN {X 0,Y 254.358,Z 744.408,A -85,B 0,C 180,E1 827.617,E2 827.617} C_VEL
